LIN {X 0,Y 418.252,Z 144.006,A -85,B 0,C 180,E1 -10131.558,E2 -10131.558} C_VEL
LIN {X 0,Y 418.26,Z 144.01,A -85,B 0,C 180,E1 -10135.159,E2 -10135.159} C_VEL
LIN {X 0,Y 418.268,Z 144.145,A -85,B 0,C 180,E1 -10137.972,E2 -10137.972} C_VEL
LIN {X 0,Y 421.832,Z 158.166,A -85,B 0,C 180,E1 -10140.894,E2 -10140.894} C_VEL
LIN {X 0,Y 424.172,Z 168.884,A -85,B 0,C 180,E1 -10142.964,E2 -10142.964} C_VEL
LIN {X 0,Y 426.899,Z 180.828,A -85,B 0,C 180,E1 -10143.399,E2 -10143.399} C_VEL
LIN {X 0,Y 430.73,Z 200.296,A -85,B 0,C 180,E1 -10144.007,E2 -10144.007} C_VEL
LIN {X 0,Y 428.4,Z 334.091,A -85,B 0,C 180,E1 -10146.301,E2 -10146.301} C_VEL
LIN {X 0,Y 427.722,Z 349.611,A -85,B 0,C 180,E1 -10146.742,E2 -10146.742} C_VEL
LIN {X 0,Y 426.907,Z 363.658,A -85,B 0,C 180,E1 -10147.324,E2 -10147.324} C_VEL
LIN {X 0,Y 425.923,Z 377.546,A -85,B 0,C 180,E1 -10148.079,E2 -10148.079} C_VEL
LIN {X 0,Y 424.665,Z 391.423,A -85,B 0,C 180,E1 -10149.03,E2 -10149.03} C_VEL
LIN {X 0,Y 423.505,Z 404.135,A -85,B 0,C 180,E1 -10150.111,E2 -10150.111} C_VEL
LIN {X 0,Y 422.222,Z 416.989,A -85,B 0,C 180,E1 -10151.437,E2 -10151.437} C_VEL
LIN {X 0,Y 421.112,Z 427.749,A -85,B 0,C 180,E1 -10152.768,E2 -10152.768} C_VEL
LIN {X 0,Y 420.039,Z 437.702,A -85,B 0,C 180,E1 -10154.223,E2 -10154.223} C_VEL
LIN {X 0,Y 419.06,Z 447.438,A -85,B 0,C 180,E1 -10155.926,E2 -10155.926} C_VEL
LIN {X 0,Y 418.334,Z 455.561,A -85,B 0,C 180,E1 -10157.631,E2 -10157.631} C_VEL
LIN {X 0,Y 417.774,Z 462.273,A -85,B 0,C 180,E1 -10159.336,E2 -10159.336} C_VEL
LIN {X 0,Y 417.406,Z 468.473,A -85,B 0,C 180,E1 -10161.284,E2 -10161.284} C_VEL
LIN {X 0,Y 417.166,Z 473.266,A -85,B 0,C 180,E1 -10163.227,E2 -10163.227} C_VEL
LIN {X 0,Y 417.051,Z 476.778,A -85,B 0,C 180,E1 -10165.167,E2 -10165.167} C_VEL
LIN {X 0,Y 416.969,Z 479.087,A -85,B 0,C 180,E1 -10167.102,E2 -10167.102} C_VEL
LIN {X 0,Y 416.989,Z 480.248,A -85,B 0,C 180,E1 -10169.034,E2 -10169.034} C_VEL
LIN {X 0,Y 416.989,Z 480.247,A -85,B 0,C 180,E1 -10170.966,E2 -10170.966} C_VEL
LIN {X 0,Y 416.969,Z 479.078,A -85,B 0,C 180,E1 -10172.898,E2 -10172.898} C_VEL
LIN {X 0,Y 417.055,Z 476.766,A -85,B 0,C 180,E1 -10174.833,E2 -10174.833} C_VEL
LIN {X 0,Y 417.224,Z 473.257,A -85,B 0,C 180,E1 -10176.772,E2 -10176.772} C_VEL
LIN {X 0,Y 417.406,Z 468.462,A -85,B 0,C 180,E1 -10178.716,E2 -10178.716} C_VEL
LIN {X 0,Y 417.774,Z 462.25,A -85,B 0,C 180,E1 -10180.664,E2 -10180.664} C_VEL
LIN {X 0,Y 418.325,Z 455.532,A -85,B 0,C 180,E1 -10182.369,E2 -10182.369} C_VEL
LIN {X 0,Y 419.17,Z 446.15,A -85,B 0,C 180,E1 -10184.318,E2 -10184.318} C_VEL
LIN {X 0,Y 420.2,Z 436.15,A -85,B 0,C 180,E1 -10186.02,E2 -10186.02} C_VEL
LIN {X 0,Y 421.313,Z 425.92,A -85,B 0,C 180,E1 -10187.473,E2 -10187.473} C_VEL
LIN {X 0,Y 422.432,Z 414.801,A -85,B 0,C 180,E1 -10188.805,E2 -10188.805} C_VEL
LIN {X 0,Y 423.625,Z 402.782,A -85,B 0,C 180,E1 -10190.009,E2 -10190.009} C_VEL
LIN {X 0,Y 424.808,Z 389.749,A -85,B 0,C 180,E1 -10191.09,E2 -10191.09} C_VEL
LIN {X 0,Y 426.096,Z 375.444,A -85,B 0,C 180,E1 -10192.039,E2 -10192.039} C_VEL
LIN {X 0,Y 427.014,Z 361.163,A -85,B 0,C 180,E1 -10192.786,E2 -10192.786} C_VEL
LIN {X 0,Y 427.86,Z 345.756,A -85,B 0,C 180,E1 -10193.378,E2 -10193.378} C_VEL
LIN {X 0,Y 428.437,Z 330.738,A -85,B 0,C 180,E1 -10193.761,E2 -10193.761} C_VEL
LIN {X 0,Y 430.681,Z 199.743,A -85,B 0,C 180,E1 -10195.998,E2 -10195.998} C_VEL
LIN {X 0,Y 424.482,Z 170.317,A -85,B 0,C 180,E1 -10196.951,E2 -10196.951} C_VEL
LIN {X 0,Y 424.129,Z 168.838,A -85,B 0,C 180,E1 -10197.034,E2 -10197.034} C_VEL
LIN {X 0,Y 421.815,Z 158.115,A -85,B 0,C 180,E1 -10199.108,E2 -10199.108} C_VEL
LIN {X 0,Y 418.268,Z 144.112,A -85,B 0,C 180,E1 -10202.028,E2 -10202.028} C_VEL
LIN {X 0,Y 418.259,Z 144.01,A -85,B 0,C 180,E1 -10204.841,E2 -10204.841} C_VEL
LIN {X 0,Y 418.251,Z 144.005,A -85,B 0,C 180,E1 -10208.442,E2 -10208.442} C_VEL
LIN {X 0,Y 418.24,Z 144.008,A -85,B 0,C 180,E1 -10212.233,E2 -10212.233} C_VEL
LIN {X 0,Y 418.236,Z 144.004,A -85,B 0,C 180,E1 -10215.109,E2 -10215.109} C_VEL
LIN {X 0,Y 418.24,Z 144.004,A -85,B 0,C 180,E1 -10217.767,E2 -10217.767} C_VEL
LIN {X 0,Y 418.253,Z 143.996,A -85,B 0,C 180,E1 -10220.62,E2 -10220.62} C_VEL
LIN {X 0,Y 418.243,Z 144.006,A -85,B 0,C 180,E1 -10223.976,E2 -10223.976} C_VEL
LIN {X 0,Y 418.243,Z 143.976,A -85,B 0,C 180,E1 -10227.472,E2 -10227.472} C_VEL
LIN {X 0,Y 418.269,Z 144.006,A -85,B 0,C 180,E1 -10230.896,E2 -10230.896} C_VEL
LIN {X 0,Y 418.27,Z 143.998,A -85,B 0,C 180,E1 -10234.096,E2 -10234.096} C_VEL
LIN {X 0,Y 418.239,Z 144.01,A -85,B 0,C 180,E1 -10237.264,E2 -10237.264} C_VEL
LIN {X 0,Y 418.284,Z 144,A -85,B 0,C 180,E1 -10240.364,E2 -10240.364} C_VEL
LIN {X 0,Y 418.317,Z 143.993,A -85,B 0,C 180,E1 -10243.405,E2 -10243.405} C_VEL
LIN {X 0,Y 418.348,Z 144.002,A -85,B 0,C 180,E1 -10246.999,E2 -10246.999} C_VEL
LIN {X 0,Y 418.34,Z 143.986,A -85,B 0,C 180,E1 -10250.329,E2 -10250.329} C_VEL
LIN {X 0,Y 418.462,Z 143.982,A -85,B 0,C 180,E1 -10253.249,E2 -10253.249} C_VEL
LIN {X 0,Y 418.334,Z 143.989,A -85,B 0,C 180,E1 -10255.182,E2 -10255.182} C_VEL
LIN {X 0,Y 418.543,Z 143.966,A -85,B 0,C 180,E1 -10258.076,E2 -10258.076} C_VEL
LIN {X 0,Y 418.668,Z 143.956,A -85,B 0,C 180,E1 -10260,E2 -10260} C_VEL
LIN {X 0,Y 418.488,Z 143.969,A -85,B 0,C 180,E1 -10262.888,E2 -10262.888} C_VEL
LIN {X 0,Y 418.459,Z 143.979,A -85,B 0,C 180,E1 -10266.516,E2 -10266.516} C_VEL
LIN {X 0,Y 418.34,Z 143.99,A -85,B 0,C 180,E1 -10269.672,E2 -10269.672} C_VEL
LIN {X 0,Y 418.348,Z 143.992,A -85,B 0,C 180,E1 -10273.001,E2 -10273.001} C_VEL
LIN {X 0,Y 418.306,Z 144.002,A -85,B 0,C 180,E1 -10276.732,E2 -10276.732} C_VEL
LIN {X 0,Y 418.272,Z 143.998,A -85,B 0,C 180,E1 -10279.79,E2 -10279.79} C_VEL
LIN {X 0,Y 418.229,Z 144.011,A -85,B 0,C 180,E1 -10282.737,E2 -10282.737} C_VEL
LIN {X 0,Y 418.226,Z 144.007,A -85,B 0,C 180,E1 -10285.907,E2 -10285.907} C_VEL
LIN {X 0,Y 418.26,Z 144.007,A -85,B 0,C 180,E1 -10289.162,E2 -10289.162} C_VEL
LIN {X 0,Y 418.251,Z 143.974,A -85,B 0,C 180,E1 -10292.842,E2 -10292.842} C_VEL
LIN {X 0,Y 418.244,Z 144.011,A -85,B 0,C 180,E1 -10296.238,E2 -10296.238} C_VEL
LIN {X 0,Y 418.2,Z 143.987,A -85,B 0,C 180,E1 -10299.688,E2 -10299.688} C_VEL
LIN {X 0,Y 418.208,Z 144.011,A -85,B 0,C 180,E1 -10302.318,E2 -10302.318} C_VEL
LIN {X 0,Y 418.236,Z 144.002,A -85,B 0,C 180,E1 -10305.109,E2 -10305.109} C_VEL
LIN {X 0,Y 418.219,Z 144.015,A -85,B 0,C 180,E1 -10307.764,E2 -10307.764} C_VEL
LIN {X 0,Y 418.238,Z 144.013,A -85,B 0,C 180,E1 -10311.557,E2 -10311.557} C_VEL
LIN {X 0,Y 418.251,Z 144.014,A -85,B 0,C 180,E1 -10315.158,E2 -10315.158} C_VEL
LIN {X 0,Y 418.24,Z 144.014,A -85,B 0,C 180,E1 -10317.471,E2 -10317.471} C_VEL
LIN {X 0,Y 418.236,Z 144.048,A -85,B 0,C 180,E1 -10319.072,E2 -10319.072} C_VEL
LIN {X 0,Y 418.652,Z 145.744,A -85,B 0,C 180,E1 -10319.519,E2 -10319.519} C_VEL
LIN {X 0,Y 421.734,Z 158.326,A -85,B 0,C 180,E1 -10322.186,E2 -10322.186} C_VEL
LIN {X 0,Y 422.604,Z 162.134,A -85,B 0,C 180,E1 -10322.921,E2 -10322.921} C_VEL
LIN {X 0,Y 426.969,Z 173.061,A -85,B 0,C 180,E1 -10323.446,E2 -10323.446} C_VEL
LIN {X 0,Y 430.77,Z 191.061,A -85,B 0,C 180,E1 -10324.027,E2 -10324.027} C_VEL
LIN {X 0,Y 428.844,Z 307.257,A -85,B 0,C 180,E1 -10326.006,E2 -10326.006} C_VEL
LIN {X 0,Y 428.375,Z 329.622,A -85,B 0,C 180,E1 -10326.428,E2 -10326.428} C_VEL
LIN {X 0,Y 427.679,Z 344.966,A -85,B 0,C 180,E1 -10326.901,E2 -10326.901} C_VEL
LIN {X 0,Y 426.893,Z 359.501,A -85,B 0,C 180,E1 -10327.544,E2 -10327.544} C_VEL
LIN {X 0,Y 425.872,Z 373.217,A -85,B 0,C 180,E1 -10328.331,E2 -10328.331} C_VEL
LIN {X 0,Y 424.685,Z 386.502,A -85,B 0,C 180,E1 -10329.284,E2 -10329.284} C_VEL
LIN {X 0,Y 423.406,Z 400.005,A -85,B 0,C 180,E1 -10330.485,E2 -10330.485} C_VEL
LIN {X 0,Y 422.251,Z 411.523,A -85,B 0,C 180,E1 -10331.727,E2 -10331.727} C_VEL
LIN {X 0,Y 421.139,Z 421.713,A -85,B 0,C 180,E1 -10333.03,E2 -10333.03} C_VEL
LIN {X 0,Y 420.108,Z 425.828,A -85,B 0,C 180,E1 -10333.591,E2 -10333.591} C_VEL
LIN {X 0,Y 416.611,Z 432.311,A -85,B 0,C 180,E1 -10334.503,E2 -10334.503} C_VEL
LIN {X 0,Y 413.133,Z 438.422,A -85,B 0,C 180,E1 -10335.477,E2 -10335.477} C_VEL
LIN {X 0,Y 412.145,Z 441.818,A -85,B 0,C 180,E1 -10336.129,E2 -10336.129} C_VEL
LIN {X 0,Y 411.461,Z 449.785,A -85,B 0,C 180,E1 -10337.922,E2 -10337.922} C_VEL
LIN {X 0,Y 410.786,Z 456.159,A -85,B 0,C 180,E1 -10339.651,E2 -10339.651} C_VEL
LIN {X 0,Y 410.382,Z 462.015,A -85,B 0,C 180,E1 -10341.63,E2 -10341.63} C_VEL
LIN {X 0,Y 410.106,Z 466.665,A -85,B 0,C 180,E1 -10343.694,E2 -10343.694} C_VEL
LIN {X 0,Y 410.013,Z 468.998,A -85,B 0,C 180,E1 -10345.083,E2 -10345.083} C_VEL
LIN {X 0,Y 409.92,Z 471.324,A -85,B 0,C 180,E1 -10347.052,E2 -10347.052} C_VEL
LIN {X 0,Y 409.917,Z 472.513,A -85,B 0,C 180,E1 -10349.018,E2 -10349.018} C_VEL
LIN {X 0,Y 409.917,Z 472.529,A -85,B 0,C 180,E1 -10350.982,E2 -10350.982} C_VEL
LIN {X 0,Y 409.92,Z 471.405,A -85,B 0,C 180,E1 -10352.948,E2 -10352.948} C_VEL
LIN {X 0,Y 410.004,Z 469.143,A -85,B 0,C 180,E1 -10354.917,E2 -10354.917} C_VEL
LIN {X 0,Y 410.113,Z 465.687,A -85,B 0,C 180,E1 -10356.89,E2 -10356.89} C_VEL
LIN {X 0,Y 410.441,Z 460.957,A -85,B 0,C 180,E1 -10358.865,E2 -10358.865} C_VEL
LIN {X 0,Y 410.894,Z 454.829,A -85,B 0,C 180,E1 -10360.845,E2 -10360.845} C_VEL
LIN {X 0,Y 411.543,Z 448.17,A -85,B 0,C 180,E1 -10362.576,E2 -10362.576} C_VEL
LIN {X 0,Y 412.45,Z 438.891,A -85,B 0,C 180,E1 -10364.557,E2 -10364.557} C_VEL
LIN {X 0,Y 413.564,Z 428.987,A -85,B 0,C 180,E1 -10366.284,E2 -10366.284} C_VEL
LIN {X 0,Y 414.74,Z 418.833,A -85,B 0,C 180,E1 -10367.759,E2 -10367.759} C_VEL
LIN {X 0,Y 416.013,Z 406.748,A -85,B 0,C 180,E1 -10369.234,E2 -10369.234} C_VEL
LIN {X 0,Y 417.297,Z 394.633,A -85,B 0,C 180,E1 -10370.455,E2 -10370.455} C_VEL
LIN {X 0,Y 418.547,Z 381.471,A -85,B 0,C 180,E1 -10371.55,E2 -10371.55} C_VEL
LIN {X 0,Y 419.642,Z 368.934,A -85,B 0,C 180,E1 -10372.396,E2 -10372.396} C_VEL
LIN {X 0,Y 420.635,Z 354.753,A -85,B 0,C 180,E1 -10373.16,E2 -10373.16} C_VEL
LIN {X 0,Y 421.407,Z 340.861,A -85,B 0,C 180,E1 -10373.725,E2 -10373.725} C_VEL
LIN {X 0,Y 422.025,Z 325.906,A -85,B 0,C 180,E1 -10374.145,E2 -10374.145} C_VEL
LIN {X 0,Y 424.493,Z 192.916,A -85,B 0,C 180,E1 -10376.453,E2 -10376.453} C_VEL
LIN {X 0,Y 420.689,Z 174.699,A -85,B 0,C 180,E1 -10377.053,E2 -10377.053} C_VEL
LIN {X 0,Y 415.364,Z 162.13,A -85,B 0,C 180,E1 -10377.699,E2 -10377.699} C_VEL
LIN {X 0,Y 412.224,Z 148.968,A -85,B 0,C 180,E1 -10380.479,E2 -10380.479} C_VEL
LIN {X 0,Y 411.237,Z 145.352,A -85,B 0,C 180,E1 -10381.296,E2 -10381.296} C_VEL
LIN {X 0,Y 411.152,Z 144.881,A -85,B 0,C 180,E1 -10381.594,E2 -10381.594} C_VEL
LIN {X 0,Y 411.202,Z 144.891,A -85,B 0,C 180,E1 -10384.876,E2 -10384.876} C_VEL
LIN {X 0,Y 411.191,Z 144.891,A -85,B 0,C 180,E1 -10388.166,E2 -10388.166} C_VEL
LIN {X 0,Y 411.161,Z 144.894,A -85,B 0,C 180,E1 -10391.808,E2 -10391.808} C_VEL
LIN {X 0,Y 411.174,Z 144.89,A -85,B 0,C 180,E1 -10395.509,E2 -10395.509} C_VEL
LIN {X 0,Y 411.148,Z 144.874,A -85,B 0,C 180,E1 -10398.775,E2 -10398.775} C_VEL
LIN {X 0,Y 411.186,Z 144.88,A -85,B 0,C 180,E1 -10402.025,E2 -10402.025} C_VEL
LIN {X 0,Y 411.204,Z 144.881,A -85,B 0,C 180,E1 -10405.123,E2 -10405.123} C_VEL
LIN {X 0,Y 411.164,Z 144.853,A -85,B 0,C 180,E1 -10408.002,E2 -10408.002} C_VEL
LIN {X 0,Y 411.177,Z 144.888,A -85,B 0,C 180,E1 -10411.407,E2 -10411.407} C_VEL
LIN {X 0,Y 411.19,Z 144.879,A -85,B 0,C 180,E1 -10414.941,E2 -10414.941} C_VEL
LIN {X 0,Y 411.205,Z 144.89,A -85,B 0,C 180,E1 -10417.913,E2 -10417.913} C_VEL
LIN {X 0,Y 411.217,Z 144.879,A -85,B 0,C 180,E1 -10421.051,E2 -10421.051} C_VEL
LIN {X 0,Y 411.212,Z 144.882,A -85,B 0,C 180,E1 -10424.13,E2 -10424.13} C_VEL
LIN {X 0,Y 411.305,Z 144.869,A -85,B 0,C 180,E1 -10427.166,E2 -10427.166} C_VEL
LIN {X 0,Y 411.292,Z 144.869,A -85,B 0,C 180,E1 -10430.161,E2 -10430.161} C_VEL
LIN {X 0,Y 411.426,Z 144.854,A -85,B 0,C 180,E1 -10433.132,E2 -10433.132} C_VEL
LIN {X 0,Y 411.3,Z 144.875,A -85,B 0,C 180,E1 -10435.099,E2 -10435.099} C_VEL
LIN {X 0,Y 411.507,Z 144.838,A -85,B 0,C 180,E1 -10438.042,E2 -10438.042} C_VEL
LIN {X 0,Y 411.636,Z 144.833,A -85,B 0,C 180,E1 -10440,E2 -10440} C_VEL
LIN {X 0,Y 411.451,Z 144.847,A -85,B 0,C 180,E1 -10442.937,E2 -10442.937} C_VEL
LIN {X 0,Y 411.426,Z 144.859,A -85,B 0,C 180,E1 -10446.867,E2 -10446.867} C_VEL
LIN {X 0,Y 411.293,Z 144.864,A -85,B 0,C 180,E1 -10449.839,E2 -10449.839} C_VEL
LIN {X 0,Y 411.308,Z 144.878,A -85,B 0,C 180,E1 -10453.104,E2 -10453.104} C_VEL
LIN {X 0,Y 411.259,Z 144.875,A -85,B 0,C 180,E1 -10456.889,E2 -10456.889} C_VEL
LIN {X 0,Y 411.232,Z 144.878,A -85,B 0,C 180,E1 -10459.987,E2 -10459.987} C_VEL
LIN {X 0,Y 411.197,Z 144.891,A -85,B 0,C 180,E1 -10463.148,E2 -10463.148} C_VEL
LIN {X 0,Y 411.235,Z 144.874,A -85,B 0,C 180,E1 -10466.381,E2 -10466.381} C_VEL
LIN {X 0,Y 411.202,Z 144.884,A -85,B 0,C 180,E1 -10469.712,E2 -10469.712} C_VEL
LIN {X 0,Y 411.205,Z 144.85,A -85,B 0,C 180,E1 -10473.156,E2 -10473.156} C_VEL
LIN {X 0,Y 411.193,Z 144.891,A -85,B 0,C 180,E1 -10476.552,E2 -10476.552} C_VEL
LIN {X 0,Y 411.213,Z 144.866,A -85,B 0,C 180,E1 -10479.728,E2 -10479.728} C_VEL
LIN {X 0,Y 411.174,Z 144.892,A -85,B 0,C 180,E1 -10483.133,E2 -10483.133} C_VEL
LIN {X 0,Y 411.168,Z 144.876,A -85,B 0,C 180,E1 -10485.881,E2 -10485.881} C_VEL
LIN {X 0,Y 411.164,Z 144.892,A -85,B 0,C 180,E1 -10488.771,E2 -10488.771} C_VEL
LIN {X 0,Y 411.196,Z 144.89,A -85,B 0,C 180,E1 -10492.026,E2 -10492.026} C_VEL
LIN {X 0,Y 411.207,Z 144.89,A -85,B 0,C 180,E1 -10495.666,E2 -10495.666} C_VEL
LIN {X 0,Y 411.224,Z 145.01,A -85,B 0,C 180,E1 -10497.537,E2 -10497.537} C_VEL
LIN {X 0,Y 414.354,Z 157.383,A -85,B 0,C 180,E1 -10500.184,E2 -10500.184} C_VEL
LIN {X 0,Y 417.031,Z 168.833,A -85,B 0,C 180,E1 -10502.464,E2 -10502.464} C_VEL
LIN {X 0,Y 418.721,Z 173.884,A -85,B 0,C 180,E1 -10502.707,E2 -10502.707} C_VEL
LIN {X 0,Y 424.313,Z 200.872,A -85,B 0,C 180,E1 -10503.596,E2 -10503.596} C_VEL
LIN {X 0,Y 421.943,Z 332.536,A -85,B 0,C 180,E1 -10505.883,E2 -10505.883} C_VEL
LIN {X 0,Y 421.314,Z 347.724,A -85,B 0,C 180,E1 -10506.302,E2 -10506.302} C_VEL
LIN {X 0,Y 420.419,Z 362.017,A -85,B 0,C 180,E1 -10506.875,E2 -10506.875} C_VEL
LIN {X 0,Y 419.503,Z 375.496,A -85,B 0,C 180,E1 -10507.596,E2 -10507.596} C_VEL
LIN {X 0,Y 418.209,Z 389.779,A -85,B 0,C 180,E1 -10508.561,E2 -10508.561} C_VEL
LIN {X 0,Y 416.935,Z 402.78,A -85,B 0,C 180,E1 -10509.656,E2 -10509.656} C_VEL
LIN {X 0,Y 415.649,Z 414.783,A -85,B 0,C 180,E1 -10510.877,E2 -10510.877} C_VEL
LIN {X 0,Y 414.492,Z 425.899,A -85,B 0,C 180,E1 -10512.23,E2 -10512.23} C_VEL
LIN {X 0,Y 413.326,Z 436.124,A -85,B 0,C 180,E1 -10513.706,E2 -10513.706} C_VEL
LIN {X 0,Y 412.275,Z 446.117,A -85,B 0,C 180,E1 -10515.437,E2 -10515.437} C_VEL
LIN {X 0,Y 411.337,Z 455.495,A -85,B 0,C 180,E1 -10517.418,E2 -10517.418} C_VEL
LIN {X 0,Y 410.763,Z 462.208,A -85,B 0,C 180,E1 -10519.152,E2 -10519.152} C_VEL
LIN {X 0,Y 410.331,Z 468.407,A -85,B 0,C 180,E1 -10521.133,E2 -10521.133} C_VEL
LIN {X 0,Y 410.082,Z 473.2,A -85,B 0,C 180,E1 -10523.11,E2 -10523.11} C_VEL
LIN {X 0,Y 409.963,Z 476.712,A -85,B 0,C 180,E1 -10525.083,E2 -10525.083} C_VEL
LIN {X 0,Y 409.867,Z 479.02,A -85,B 0,C 180,E1 -10527.051,E2 -10527.051} C_VEL
LIN {X 0,Y 409.915,Z 480.182,A -85,B 0,C 180,E1 -10529.018,E2 -10529.018} C_VEL
LIN {X 0,Y 409.915,Z 480.181,A -85,B 0,C 180,E1 -10530.982,E2 -10530.982} C_VEL
LIN {X 0,Y 409.867,Z 479.012,A -85,B 0,C 180,E1 -10532.949,E2 -10532.949} C_VEL
LIN {X 0,Y 409.968,Z 476.699,A -85,B 0,C 180,E1 -10534.917,E2 -10534.917} C_VEL
LIN {X 0,Y 410.155,Z 473.19,A -85,B 0,C 180,E1 -10536.889,E2 -10536.889} C_VEL
LIN {X 0,Y 410.331,Z 468.394,A -85,B 0,C 180,E1 -10538.867,E2 -10538.867} C_VEL
LIN {X 0,Y 410.763,Z 462.183,A -85,B 0,C 180,E1 -10540.848,E2 -10540.848} C_VEL
LIN {X 0,Y 411.33,Z 455.464,A -85,B 0,C 180,E1 -10542.583,E2 -10542.583} C_VEL
LIN {X 0,Y 412.263,Z 446.081,A -85,B 0,C 180,E1 -10544.563,E2 -10544.563} C_VEL
LIN {X 0,Y 413.301,Z 436.081,A -85,B 0,C 180,E1 -10546.295,E2 -10546.295} C_VEL
LIN {X 0,Y 414.588,Z 424.669,A -85,B 0,C 180,E1 -10547.926,E2 -10547.926} C_VEL
LIN {X 0,Y 415.901,Z 412.51,A -85,B 0,C 180,E1 -10549.368,E2 -10549.368} C_VEL
LIN {X 0,Y 417.212,Z 400.083,A -85,B 0,C 180,E1 -10550.588,E2 -10550.588} C_VEL
LIN {X 0,Y 418.48,Z 386.466,A -85,B 0,C 180,E1 -10551.683,E2 -10551.683} C_VEL
LIN {X 0,Y 419.708,Z 372.359,A -85,B 0,C 180,E1 -10552.587,E2 -10552.587} C_VEL
LIN {X 0,Y 420.673,Z 358.594,A -85,B 0,C 180,E1 -10553.274,E2 -10553.274} C_VEL
LIN {X 0,Y 421.505,Z 342.93,A -85,B 0,C 180,E1 -10553.849,E2 -10553.849} C_VEL
LIN {X 0,Y 422.007,Z 327.643,A -85,B 0,C 180,E1 -10554.211,E2 -10554.211} C_VEL
LIN {X 0,Y 424.332,Z 201.581,A -85,B 0,C 180,E1 -10556.381,E2 -10556.381} C_VEL
LIN {X 0,Y 419.585,Z 177.878,A -85,B 0,C 180,E1 -10557.147,E2 -10557.147} C_VEL
LIN {X 0,Y 417.817,Z 171.092,A -85,B 0,C 180,E1 -10557.4,E2 -10557.4} C_VEL
LIN {X 0,Y 416.985,Z 168.667,A -85,B 0,C 180,E1 -10557.548,E2 -10557.548} C_VEL
LIN {X 0,Y 414.1,Z 156.176,A -85,B 0,C 180,E1 -10560.054,E2 -10560.054} C_VEL
LIN {X 0,Y 411.224,Z 144.948,A -85,B 0,C 180,E1 -10562.481,E2 -10562.481} C_VEL
LIN {X 0,Y 411.198,Z 144.881,A -85,B 0,C 180,E1 -10565.529,E2 -10565.529} C_VEL
LIN {X 0,Y 411.212,Z 144.874,A -85,B 0,C 180,E1 -10569.225,E2 -10569.225} C_VEL
LIN {X 0,Y 411.182,Z 144.885,A -85,B 0,C 180,E1 -10572.696,E2 -10572.696} C_VEL
LIN {X 0,Y 411.168,Z 144.893,A -85,B 0,C 180,E1 -10575.881,E2 -10575.881} C_VEL
LIN {X 0,Y 411.163,Z 144.873,A -85,B 0,C 180,E1 -10578.772,E2 -10578.772} C_VEL
LIN {X 0,Y 411.205,Z 144.885,A -85,B 0,C 180,E1 -10581.832,E2 -10581.832} C_VEL
LIN {X 0,Y 411.203,Z 144.87,A -85,B 0,C 180,E1 -10585.123,E2 -10585.123} C_VEL
LIN {X 0,Y 411.164,Z 144.862,A -85,B 0,C 180,E1 -10588.003,E2 -10588.003} C_VEL
LIN {X 0,Y 411.219,Z 144.889,A -85,B 0,C 180,E1 -10591.41,E2 -10591.41} C_VEL
LIN {X 0,Y 411.238,Z 144.874,A -85,B 0,C 180,E1 -10593.619,E2 -10593.619} C_VEL
LIN {X 0,Y 411.204,Z 144.89,A -85,B 0,C 180,E1 -10596.853,E2 -10596.853} C_VEL
LIN {X 0,Y 411.216,Z 144.88,A -85,B 0,C 180,E1 -10600.051,E2 -10600.051} C_VEL
LIN {X 0,Y 411.264,Z 144.874,A -85,B 0,C 180,E1 -10603.131,E2 -10603.131} C_VEL
LIN {X 0,Y 411.307,Z 144.878,A -85,B 0,C 180,E1 -10606.896,E2 -10606.896} C_VEL
LIN {X 0,Y 411.292,Z 144.864,A -85,B 0,C 180,E1 -10610.161,E2 -10610.161} C_VEL
LIN {X 0,Y 411.426,Z 144.859,A -85,B 0,C 180,E1 -10613.133,E2 -10613.133} C_VEL
LIN {X 0,Y 411.305,Z 144.865,A -85,B 0,C 180,E1 -10615.099,E2 -10615.099} C_VEL
LIN {X 0,Y 411.511,Z 144.842,A -85,B 0,C 180,E1 -10618.043,E2 -10618.043} C_VEL
LIN {X 0,Y 411.637,Z 144.832,A -85,B 0,C 180,E1 -10620,E2 -10620} C_VEL
LIN {X 0,Y 411.445,Z 144.846,A -85,B 0,C 180,E1 -10622.937,E2 -10622.937} C_VEL
LIN {X 0,Y 411.424,Z 144.855,A -85,B 0,C 180,E1 -10626.514,E2 -10626.514} C_VEL
LIN {X 0,Y 411.292,Z 144.869,A -85,B 0,C 180,E1 -10629.839,E2 -10629.839} C_VEL
LIN {X 0,Y 411.307,Z 144.869,A -85,B 0,C 180,E1 -10633.104,E2 -10633.104} C_VEL
LIN {X 0,Y 411.258,Z 144.879,A -85,B 0,C 180,E1 -10636.889,E2 -10636.889} C_VEL
LIN {X 0,Y 411.232,Z 144.874,A -85,B 0,C 180,E1 -10639.987,E2 -10639.987} C_VEL
LIN {X 0,Y 411.19,Z 144.888,A -85,B 0,C 180,E1 -10643.148,E2 -10643.148} C_VEL
LIN {X 0,Y 411.176,Z 144.889,A -85,B 0,C 180,E1 -10646.385,E2 -10646.385} C_VEL
LIN {X 0,Y 411.198,Z 144.876,A -85,B 0,C 180,E1 -10649.713,E2 -10649.713} C_VEL
LIN {X 0,Y 411.205,Z 144.854,A -85,B 0,C 180,E1 -10653.156,E2 -10653.156} C_VEL
LIN {X 0,Y 411.192,Z 144.889,A -85,B 0,C 180,E1 -10656.552,E2 -10656.552} C_VEL
LIN {X 0,Y 411.169,Z 144.862,A -85,B 0,C 180,E1 -10659.72,E2 -10659.72} C_VEL
LIN {X 0,Y 411.163,Z 144.894,A -85,B 0,C 180,E1 -10663.135,E2 -10663.135} C_VEL
LIN {X 0,Y 411.164,Z 144.876,A -85,B 0,C 180,E1 -10665.882,E2 -10665.882} C_VEL
LIN {X 0,Y 411.148,Z 144.896,A -85,B 0,C 180,E1 -10668.774,E2 -10668.774} C_VEL
LIN {X 0,Y 411.186,Z 144.891,A -85,B 0,C 180,E1 -10672.025,E2 -10672.025} C_VEL
LIN {X 0,Y 411.203,Z 144.892,A -85,B 0,C 180,E1 -10675.123,E2 -10675.123} C_VEL
LIN {X 0,Y 411.153,Z 144.882,A -85,B 0,C 180,E1 -10678.405,E2 -10678.405} C_VEL
LIN {X 0,Y 411.218,Z 145.209,A -85,B 0,C 180,E1 -10678.763,E2 -10678.763} C_VEL
LIN {X 0,Y 414.2,Z 156.981,A -85,B 0,C 180,E1 -10681.358,E2 -10681.358} C_VEL
LIN {X 0,Y 415.438,Z 162.329,A -85,B 0,C 180,E1 -10682.423,E2 -10682.423} C_VEL
LIN {X 0,Y 420.788,Z 175.035,A -85,B 0,C 180,E1 -10683.06,E2 -10683.06} C_VEL
LIN {X 0,Y 424.408,Z 192.602,A -85,B 0,C 180,E1 -10683.634,E2 -10683.634} C_VEL
LIN {X 0,Y 422.385,Z 307.349,A -85,B 0,C 180,E1 -10685.616,E2 -10685.616} C_VEL
LIN {X 0,Y 421.877,Z 329.705,A -85,B 0,C 180,E1 -10686.042,E2 -10686.042} C_VEL
LIN {X 0,Y 421.187,Z 344.47,A -85,B 0,C 180,E1 -10686.499,E2 -10686.499} C_VEL
LIN {X 0,Y 420.4,Z 358.732,A -85,B 0,C 180,E1 -10687.129,E2 -10687.129} C_VEL
LIN {X 0,Y 419.42,Z 371.398,A -85,B 0,C 180,E1 -10687.851,E2 -10687.851} C_VEL
LIN {X 0,Y 418.161,Z 385.01,A -85,B 0,C 180,E1 -10688.817,E2 -10688.817} C_VEL
LIN {X 0,Y 416.821,Z 398.82,A -85,B 0,C 180,E1 -10690.036,E2 -10690.036} C_VEL
LIN {X 0,Y 415.605,Z 410.212,A -85,B 0,C 180,E1 -10691.259,E2 -10691.259} C_VEL
LIN {X 0,Y 414.324,Z 421.713,A -85,B 0,C 180,E1 -10692.732,E2 -10692.732} C_VEL
LIN {X 0,Y 413.292,Z 431.392,A -85,B 0,C 180,E1 -10694.212,E2 -10694.212} C_VEL
LIN {X 0,Y 412.229,Z 440.881,A -85,B 0,C 180,E1 -10695.94,E2 -10695.94} C_VEL
LIN {X 0,Y 412.145,Z 441.818,A -85,B 0,C 180,E1 -10696.129,E2 -10696.129} C_VEL
LIN {X 0,Y 411.184,Z 445.107,A -85,B 0,C 180,E1 -10696.8,E2 -10696.8} C_VEL
LIN {X 0,Y 407.838,Z 450.165,A -85,B 0,C 180,E1 -10697.9,E2 -10697.9} C_VEL
LIN {X 0,Y 404.548,Z 454.796,A -85,B 0,C 180,E1 -10699.055,E2 -10699.055} C_VEL
LIN {X 0,Y 403.691,Z 457.295,A -85,B 0,C 180,E1 -10699.804,E2 -10699.804} C_VEL
LIN {X 0,Y 403.32,Z 462.082,A -85,B 0,C 180,E1 -10701.482,E2 -10701.482} C_VEL
LIN {X 0,Y 403.076,Z 465.55,A -85,B 0,C 180,E1 -10702.99,E2 -10702.99} C_VEL
LIN {X 0,Y 402.928,Z 469.065,A -85,B 0,C 180,E1 -10704.997,E2 -10704.997} C_VEL
LIN {X 0,Y 402.819,Z 471.391,A -85,B 0,C 180,E1 -10707,E2 -10707} C_VEL
LIN {X 0,Y 402.845,Z 472.579,A -85,B 0,C 180,E1 -10709,E2 -10709} C_VEL
LIN {X 0,Y 402.846,Z 472.595,A -85,B 0,C 180,E1 -10711,E2 -10711} C_VEL
LIN {X 0,Y 402.819,Z 471.472,A -85,B 0,C 180,E1 -10713,E2 -10713} C_VEL
LIN {X 0,Y 402.917,Z 469.209,A -85,B 0,C 180,E1 -10715.003,E2 -10715.003} C_VEL
LIN {X 0,Y 403.048,Z 465.753,A -85,B 0,C 180,E1 -10717.011,E2 -10717.011} C_VEL
LIN {X 0,Y 403.403,Z 461.022,A -85,B 0,C 180,E1 -10719.021,E2 -10719.021} C_VEL
LIN {X 0,Y 403.889,Z 454.894,A -85,B 0,C 180,E1 -10721.035,E2 -10721.035} C_VEL
LIN {X 0,Y 404.538,Z 448.235,A -85,B 0,C 180,E1 -10722.797,E2 -10722.797} C_VEL
LIN {X 0,Y 405.515,Z 438.955,A -85,B 0,C 180,E1 -10724.811,E2 -10724.811} C_VEL
LIN {X 0,Y 406.713,Z 429.051,A -85,B 0,C 180,E1 -10726.566,E2 -10726.566} C_VEL
LIN {X 0,Y 407.946,Z 418.897,A -85,B 0,C 180,E1 -10728.065,E2 -10728.065} C_VEL
LIN {X 0,Y 409.148,Z 407.879,A -85,B 0,C 180,E1 -10729.439,E2 -10729.439} C_VEL
LIN {X 0,Y 410.483,Z 395.984,A -85,B 0,C 180,E1 -10730.679,E2 -10730.679} C_VEL
LIN {X 0,Y 411.774,Z 383.112,A -85,B 0,C 180,E1 -10731.791,E2 -10731.791} C_VEL
LIN {X 0,Y 413.082,Z 368.993,A -85,B 0,C 180,E1 -10732.772,E2 -10732.772} C_VEL
LIN {X 0,Y 414.153,Z 354.057,A -85,B 0,C 180,E1 -10733.582,E2 -10733.582} C_VEL
LIN {X 0,Y 414.966,Z 339.085,A -85,B 0,C 180,E1 -10734.183,E2 -10734.183} C_VEL
LIN {X 0,Y 415.583,Z 324.447,A -85,B 0,C 180,E1 -10734.577,E2 -10734.577} C_VEL
LIN {X 0,Y 418.139,Z 194.125,A -85,B 0,C 180,E1 -10736.865,E2 -10736.865} C_VEL
LIN {X 0,Y 414.702,Z 177.431,A -85,B 0,C 180,E1 -10737.425,E2 -10737.425} C_VEL
LIN {X 0,Y 408.159,Z 162.135,A -85,B 0,C 180,E1 -10738.237,E2 -10738.237} C_VEL
LIN {X 0,Y 404.958,Z 149.039,A -85,B 0,C 180,E1 -10741.085,E2 -10741.085} C_VEL
LIN {X 0,Y 404.148,Z 145.977,A -85,B 0,C 180,E1 -10741.822,E2 -10741.822} C_VEL
LIN {X 0,Y 404.138,Z 145.762,A -85,B 0,C 180,E1 -10743.813,E2 -10743.813} C_VEL
LIN {X 0,Y 404.132,Z 145.761,A -85,B 0,C 180,E1 -10746.874,E2 -10746.874} C_VEL
LIN {X 0,Y 404.118,Z 145.757,A -85,B 0,C 180,E1 -10750.075,E2 -10750.075} C_VEL
LIN {X 0,Y 404.142,Z 145.758,A -85,B 0,C 180,E1 -10753.082,E2 -10753.082} C_VEL
LIN {X 0,Y 404.121,Z 145.768,A -85,B 0,C 180,E1 -10755.922,E2 -10755.922} C_VEL
LIN {X 0,Y 404.102,Z 145.753,A -85,B 0,C 180,E1 -10758.633,E2 -10758.633} C_VEL
LIN {X 0,Y 404.14,Z 145.752,A -85,B 0,C 180,E1 -10761.495,E2 -10761.495} C_VEL
LIN {X 0,Y 404.179,Z 145.757,A -85,B 0,C 180,E1 -10764.983,E2 -10764.983} C_VEL
LIN {X 0,Y 404.138,Z 145.729,A -85,B 0,C 180,E1 -10768.443,E2 -10768.443} C_VEL
LIN {X 0,Y 404.152,Z 145.761,A -85,B 0,C 180,E1 -10770.862,E2 -10770.862} C_VEL
LIN {X 0,Y 404.155,Z 145.755,A -85,B 0,C 180,E1 -10774.722,E2 -10774.722} C_VEL
LIN {X 0,Y 404.168,Z 145.763,A -85,B 0,C 180,E1 -10777.508,E2 -10777.508} C_VEL
LIN {X 0,Y 404.162,Z 145.757,A -85,B 0,C 180,E1 -10780.707,E2 -10780.707} C_VEL
LIN {X 0,Y 404.183,Z 145.761,A -85,B 0,C 180,E1 -10783.846,E2 -10783.846} C_VEL
LIN {X 0,Y 404.285,Z 145.743,A -85,B 0,C 180,E1 -10786.939,E2 -10786.939} C_VEL
LIN {X 0,Y 404.258,Z 145.747,A -85,B 0,C 180,E1 -10789.988,E2 -10789.988} C_VEL
LIN {X 0,Y 404.371,Z 145.732,A -85,B 0,C 180,E1 -10793.012,E2 -10793.012} C_VEL
LIN {X 0,Y 404.273,Z 145.75,A -85,B 0,C 180,E1 -10795.013,E2 -10795.013} C_VEL
LIN {X 0,Y 404.475,Z 145.713,A -85,B 0,C 180,E1 -10798.008,E2 -10798.008} C_VEL
LIN {X 0,Y 404.605,Z 145.709,A -85,B 0,C 180,E1 -10800,E2 -10800} C_VEL
LIN {X 0,Y 404.409,Z 145.723,A -85,B 0,C 180,E1 -10802.988,E2 -10802.988} C_VEL
LIN {X 0,Y 404.372,Z 145.739,A -85,B 0,C 180,E1 -10806.988,E2 -10806.988} C_VEL
LIN {X 0,Y 404.258,Z 145.741,A -85,B 0,C 180,E1 -10810.012,E2 -10810.012} C_VEL
LIN {X 0,Y 404.268,Z 145.753,A -85,B 0,C 180,E1 -10813.211,E2 -10813.211} C_VEL
LIN {X 0,Y 404.218,Z 145.754,A -85,B 0,C 180,E1 -10817.007,E2 -10817.007} C_VEL
LIN {X 0,Y 404.165,Z 145.758,A -85,B 0,C 180,E1 -10820.351,E2 -10820.351} C_VEL
LIN {X 0,Y 404.161,Z 145.764,A -85,B 0,C 180,E1 -10823.575,E2 -10823.575} C_VEL
LIN {X 0,Y 404.182,Z 145.751,A -85,B 0,C 180,E1 -10825.766,E2 -10825.766} C_VEL
LIN {X 0,Y 404.196,Z 145.759,A -85,B 0,C 180,E1 -10827.999,E2 -10827.999} C_VEL
LIN {X 0,Y 404.139,Z 145.743,A -85,B 0,C 180,E1 -10831.558,E2 -10831.558} C_VEL
LIN {X 0,Y 404.179,Z 145.748,A -85,B 0,C 180,E1 -10835.017,E2 -10835.017} C_VEL
LIN {X 0,Y 404.155,Z 145.754,A -85,B 0,C 180,E1 -10838.757,E2 -10838.757} C_VEL
LIN {X 0,Y 404.123,Z 145.756,A -85,B 0,C 180,E1 -10841.599,E2 -10841.599} C_VEL
LIN {X 0,Y 404.146,Z 145.761,A -85,B 0,C 180,E1 -10844.522,E2 -10844.522} C_VEL
LIN {X 0,Y 404.137,Z 145.762,A -85,B 0,C 180,E1 -10847.295,E2 -10847.295} C_VEL
LIN {X 0,Y 404.169,Z 145.753,A -85,B 0,C 180,E1 -10849.955,E2 -10849.955} C_VEL
LIN {X 0,Y 404.138,Z 145.765,A -85,B 0,C 180,E1 -10853.125,E2 -10853.125} C_VEL
LIN {X 0,Y 404.146,Z 145.755,A -85,B 0,C 180,E1 -10856.188,E2 -10856.188} C_VEL
LIN {X 0,Y 404.224,Z 145.982,A -85,B 0,C 180,E1 -10857.119,E2 -10857.119} C_VEL
LIN {X 0,Y 407.179,Z 157.584,A -85,B 0,C 180,E1 -10859.656,E2 -10859.656} C_VEL
LIN {X 0,Y 409.765,Z 168.645,A -85,B 0,C 180,E1 -10861.922,E2 -10861.922} C_VEL
LIN {X 0,Y 412.564,Z 175.812,A -85,B 0,C 180,E1 -10862.303,E2 -10862.303} C_VEL
LIN {X 0,Y 417.739,Z 200.965,A -85,B 0,C 180,E1 -10863.15,E2 -10863.15} C_VEL
LIN {X 0,Y 417.943,Z 204.055,A -85,B 0,C 180,E1 -10863.222,E2 -10863.222} C_VEL
LIN {X 0,Y 415.445,Z 333.991,A -85,B 0,C 180,E1 -10865.514,E2 -10865.514} C_VEL
LIN {X 0,Y 414.7,Z 349.498,A -85,B 0,C 180,E1 -10865.967,E2 -10865.967} C_VEL
LIN {X 0,Y 413.793,Z 363.539,A -85,B 0,C 180,E1 -10866.563,E2 -10866.563} C_VEL
LIN {X 0,Y 412.754,Z 377.424,A -85,B 0,C 180,E1 -10867.341,E2 -10867.341} C_VEL
LIN {X 0,Y 411.41,Z 391.299,A -85,B 0,C 180,E1 -10868.32,E2 -10868.32} C_VEL
LIN {X 0,Y 410.102,Z 404.009,A -85,B 0,C 180,E1 -10869.432,E2 -10869.432} C_VEL
LIN {X 0,Y 408.686,Z 416.861,A -85,B 0,C 180,E1 -10870.799,E2 -10870.799} C_VEL
LIN {X 0,Y 407.469,Z 427.62,A -85,B 0,C 180,E1 -10872.172,E2 -10872.172} C_VEL
LIN {X 0,Y 406.289,Z 437.572,A -85,B 0,C 180,E1 -10873.674,E2 -10873.674} C_VEL
LIN {X 0,Y 405.175,Z 447.307,A -85,B 0,C 180,E1 -10875.433,E2 -10875.433} C_VEL
LIN {X 0,Y 404.36,Z 455.43,A -85,B 0,C 180,E1 -10877.197,E2 -10877.197} C_VEL
LIN {X 0,Y 403.764,Z 462.143,A -85,B 0,C 180,E1 -10878.961,E2 -10878.961} C_VEL
LIN {X 0,Y 403.277,Z 468.341,A -85,B 0,C 180,E1 -10880.976,E2 -10880.976} C_VEL
LIN {X 0,Y 403.002,Z 473.134,A -85,B 0,C 180,E1 -10882.988,E2 -10882.988} C_VEL
LIN {X 0,Y 402.879,Z 476.646,A -85,B 0,C 180,E1 -10884.996,E2 -10884.996} C_VEL
LIN {X 0,Y 402.769,Z 478.954,A -85,B 0,C 180,E1 -10886.999,E2 -10886.999} C_VEL
LIN {X 0,Y 402.842,Z 480.116,A -85,B 0,C 180,E1 -10889,E2 -10889} C_VEL
LIN {X 0,Y 402.842,Z 480.115,A -85,B 0,C 180,E1 -10891,E2 -10891} C_VEL
LIN {X 0,Y 402.769,Z 478.945,A -85,B 0,C 180,E1 -10893.001,E2 -10893.001} C_VEL
LIN {X 0,Y 402.883,Z 476.632,A -85,B 0,C 180,E1 -10895.004,E2 -10895.004} C_VEL
LIN {X 0,Y 403.065,Z 473.123,A -85,B 0,C 180,E1 -10897.011,E2 -10897.011} C_VEL
LIN {X 0,Y 403.277,Z 468.326,A -85,B 0,C 180,E1 -10899.024,E2 -10899.024} C_VEL
LIN {X 0,Y 403.763,Z 462.115,A -85,B 0,C 180,E1 -10901.038,E2 -10901.038} C_VEL
LIN {X 0,Y 404.354,Z 455.395,A -85,B 0,C 180,E1 -10902.803,E2 -10902.803} C_VEL
LIN {X 0,Y 405.162,Z 447.271,A -85,B 0,C 180,E1 -10904.567,E2 -10904.567} C_VEL
LIN {X 0,Y 406.268,Z 437.529,A -85,B 0,C 180,E1 -10906.326,E2 -10906.326} C_VEL
LIN {X 0,Y 407.474,Z 427.567,A -85,B 0,C 180,E1 -10907.827,E2 -10907.827} C_VEL
LIN {X 0,Y 408.69,Z 416.802,A -85,B 0,C 180,E1 -10909.201,E2 -10909.201} C_VEL
LIN {X 0,Y 410.107,Z 403.935,A -85,B 0,C 180,E1 -10910.567,E2 -10910.567} C_VEL
LIN {X 0,Y 411.382,Z 391.191,A -85,B 0,C 180,E1 -10911.681,E2 -10911.681} C_VEL
LIN {X 0,Y 412.752,Z 377.287,A -85,B 0,C 180,E1 -10912.659,E2 -10912.659} C_VEL
LIN {X 0,Y 413.726,Z 364.28,A -85,B 0,C 180,E1 -10913.395,E2 -10913.395} C_VEL
LIN {X 0,Y 414.728,Z 349.27,A -85,B 0,C 180,E1 -10914.031,E2 -10914.031} C_VEL
LIN {X 0,Y 415.404,Z 333.586,A -85,B 0,C 180,E1 -10914.488,E2 -10914.488} C_VEL
LIN {X 0,Y 417.753,Z 210.809,A -85,B 0,C 180,E1 -10916.654,E2 -10916.654} C_VEL
LIN {X 0,Y 417.863,Z 201.734,A -85,B 0,C 180,E1 -10916.817,E2 -10916.817} C_VEL
LIN {X 0,Y 412.298,Z 174.92,A -85,B 0,C 180,E1 -10917.723,E2 -10917.723} C_VEL
LIN {X 0,Y 409.796,Z 168.717,A -85,B 0,C 180,E1 -10918.058,E2 -10918.058} C_VEL
LIN {X 0,Y 407.182,Z 157.529,A -85,B 0,C 180,E1 -10920.345,E2 -10920.345} C_VEL
LIN {X 0,Y 404.187,Z 145.837,A -85,B 0,C 180,E1 -10922.918,E2 -10922.918} C_VEL
LIN {X 0,Y 404.143,Z 145.759,A -85,B 0,C 180,E1 -10926.246,E2 -10926.246} C_VEL
LIN {X 0,Y 404.152,Z 145.756,A -85,B 0,C 180,E1 -10928.757,E2 -10928.757} C_VEL
LIN {X 0,Y 404.123,Z 145.773,A -85,B 0,C 180,E1 -10931.6,E2 -10931.6} C_VEL
LIN {X 0,Y 404.145,Z 145.753,A -85,B 0,C 180,E1 -10934.522,E2 -10934.522} C_VEL
LIN {X 0,Y 404.136,Z 145.768,A -85,B 0,C 180,E1 -10937.296,E2 -10937.296} C_VEL
LIN {X 0,Y 404.169,Z 145.74,A -85,B 0,C 180,E1 -10939.956,E2 -10939.956} C_VEL
LIN {X 0,Y 404.136,Z 145.77,A -85,B 0,C 180,E1 -10943.125,E2 -10943.125} C_VEL
LIN {X 0,Y 404.138,Z 145.733,A -85,B 0,C 180,E1 -10946.187,E2 -10946.187} C_VEL
LIN {X 0,Y 404.146,Z 145.759,A -85,B 0,C 180,E1 -10949.715,E2 -10949.715} C_VEL
LIN {X 0,Y 404.196,Z 145.754,A -85,B 0,C 180,E1 -10953.123,E2 -10953.123} C_VEL
LIN {X 0,Y 404.179,Z 145.762,A -85,B 0,C 180,E1 -10955.335,E2 -10955.335} C_VEL
LIN {X 0,Y 404.14,Z 145.759,A -85,B 0,C 180,E1 -10958.581,E2 -10958.581} C_VEL
LIN {X 0,Y 404.205,Z 145.758,A -85,B 0,C 180,E1 -10961.762,E2 -10961.762} C_VEL
LIN {X 0,Y 404.207,Z 145.748,A -85,B 0,C 180,E1 -10964.882,E2 -10964.882} C_VEL
LIN {X 0,Y 404.258,Z 145.751,A -85,B 0,C 180,E1 -10967.959,E2 -10967.959} C_VEL
LIN {X 0,Y 404.267,Z 145.741,A -85,B 0,C 180,E1 -10970.999,E2 -10970.999} C_VEL
LIN {X 0,Y 404.395,Z 145.734,A -85,B 0,C 180,E1 -10974.015,E2 -10974.015} C_VEL
LIN {X 0,Y 404.48,Z 145.717,A -85,B 0,C 180,E1 -10978.009,E2 -10978.009} C_VEL
LIN {X 0,Y 404.607,Z 145.708,A -85,B 0,C 180,E1 -10980,E2 -10980} C_VEL
LIN {X 0,Y 404.404,Z 145.723,A -85,B 0,C 180,E1 -10982.989,E2 -10982.989} C_VEL
LIN {X 0,Y 404.373,Z 145.734,A -85,B 0,C 180,E1 -10986.509,E2 -10986.509} C_VEL
LIN {X 0,Y 404.267,Z 145.74,A -85,B 0,C 180,E1 -10989.002,E2 -10989.002} C_VEL
LIN {X 0,Y 404.257,Z 145.756,A -85,B 0,C 180,E1 -10992.042,E2 -10992.042} C_VEL
LIN {X 0,Y 404.198,Z 145.749,A -85,B 0,C 180,E1 -10995.118,E2 -10995.118} C_VEL
LIN {X 0,Y 404.202,Z 145.757,A -85,B 0,C 180,E1 -10998.239,E2 -10998.239} C_VEL
LIN {X 0,Y 404.139,Z 145.762,A -85,B 0,C 180,E1 -11001.419,E2 -11001.419} C_VEL
LIN {X 0,Y 404.149,Z 145.756,A -85,B 0,C 180,E1 -11004.668,E2 -11004.668} C_VEL
LIN {X 0,Y 404.117,Z 145.771,A -85,B 0,C 180,E1 -11008.006,E2 -11008.006} C_VEL
LIN {X 0,Y 404.144,Z 145.749,A -85,B 0,C 180,E1 -11010.285,E2 -11010.285} C_VEL
LIN {X 0,Y 404.139,Z 145.742,A -85,B 0,C 180,E1 -11013.813,E2 -11013.813} C_VEL
LIN {X 0,Y 404.135,Z 145.77,A -85,B 0,C 180,E1 -11016.875,E2 -11016.875} C_VEL
LIN {X 0,Y 404.117,Z 145.738,A -85,B 0,C 180,E1 -11020.075,E2 -11020.075} C_VEL
LIN {X 0,Y 404.143,Z 145.767,A -85,B 0,C 180,E1 -11023.082,E2 -11023.082} C_VEL
LIN {X 0,Y 404.121,Z 145.753,A -85,B 0,C 180,E1 -11025.922,E2 -11025.922} C_VEL
LIN {X 0,Y 404.103,Z 145.775,A -85,B 0,C 180,E1 -11028.633,E2 -11028.633} C_VEL
LIN {X 0,Y 404.141,Z 145.767,A -85,B 0,C 180,E1 -11031.495,E2 -11031.495} C_VEL
LIN {X 0,Y 404.174,Z 145.766,A -85,B 0,C 180,E1 -11034.983,E2 -11034.983} C_VEL
LIN {X 0,Y 404.141,Z 145.907,A -85,B 0,C 180,E1 -11038.25,E2 -11038.25} C_VEL
LIN {X 0,Y 406.612,Z 155.688,A -85,B 0,C 180,E1 -11040.498,E2 -11040.498} C_VEL
LIN {X 0,Y 408.209,Z 162.188,A -85,B 0,C 180,E1 -11041.874,E2 -11041.874} C_VEL
LIN {X 0,Y 414.812,Z 177.978,A -85,B 0,C 180,E1 -11042.694,E2 -11042.694} C_VEL
LIN {X 0,Y 418.039,Z 193.082,A -85,B 0,C 180,E1 -11043.208,E2 -11043.208} C_VEL
LIN {X 0,Y 415.95,Z 307.441,A -85,B 0,C 180,E1 -11045.213,E2 -11045.213} C_VEL
LIN {X 0,Y 415.405,Z 329.787,A -85,B 0,C 180,E1 -11045.645,E2 -11045.645} C_VEL
LIN {X 0,Y 414.67,Z 344.721,A -85,B 0,C 180,E1 -11046.115,E2 -11046.115} C_VEL
LIN {X 0,Y 413.844,Z 359.189,A -85,B 0,C 180,E1 -11046.768,E2 -11046.768} C_VEL
LIN {X 0,Y 412.85,Z 371.472,A -85,B 0,C 180,E1 -11047.479,E2 -11047.479} C_VEL
LIN {X 0,Y 411.55,Z 385.083,A -85,B 0,C 180,E1 -11048.46,E2 -11048.46} C_VEL
LIN {X 0,Y 410.245,Z 397.602,A -85,B 0,C 180,E1 -11049.571,E2 -11049.571} C_VEL
LIN {X 0,Y 408.961,Z 409.216,A -85,B 0,C 180,E1 -11050.812,E2 -11050.812} C_VEL
LIN {X 0,Y 407.755,Z 420.004,A -85,B 0,C 180,E1 -11052.186,E2 -11052.186} C_VEL
LIN {X 0,Y 406.572,Z 429.98,A -85,B 0,C 180,E1 -11053.686,E2 -11053.686} C_VEL
LIN {X 0,Y 405.422,Z 439.723,A -85,B 0,C 180,E1 -11055.442,E2 -11055.442} C_VEL
LIN {X 0,Y 404.629,Z 447.844,A -85,B 0,C 180,E1 -11057.206,E2 -11057.206} C_VEL
LIN {X 0,Y 403.913,Z 454.546,A -85,B 0,C 180,E1 -11058.966,E2 -11058.966} C_VEL
LIN {X 0,Y 403.691,Z 457.295,A -85,B 0,C 180,E1 -11059.804,E2 -11059.804} C_VEL
LIN {X 0,Y 402.872,Z 459.669,A -85,B 0,C 180,E1 -11060.564,E2 -11060.564} C_VEL
LIN {X 0,Y 399.767,Z 463.197,A -85,B 0,C 180,E1 -11061.811,E2 -11061.811} C_VEL
LIN {X 0,Y 397.172,Z 465.6,A -85,B 0,C 180,E1 -11062.839,E2 -11062.839} C_VEL
LIN {X 0,Y 396.02,Z 467.14,A -85,B 0,C 180,E1 -11063.651,E2 -11063.651} C_VEL
LIN {X 0,Y 395.904,Z 467.596,A -85,B 0,C 180,E1 -11063.929,E2 -11063.929} C_VEL
LIN {X 0,Y 395.765,Z 470.439,A -85,B 0,C 180,E1 -11065.927,E2 -11065.927} C_VEL
LIN {X 0,Y 395.759,Z 472.191,A -85,B 0,C 180,E1 -11067.965,E2 -11067.965} C_VEL
LIN {X 0,Y 395.758,Z 472.804,A -85,B 0,C 180,E1 -11070,E2 -11070} C_VEL
LIN {X 0,Y 395.759,Z 472.239,A -85,B 0,C 180,E1 -11072.035,E2 -11072.035} C_VEL
LIN {X 0,Y 395.762,Z 470.551,A -85,B 0,C 180,E1 -11074.073,E2 -11074.073} C_VEL
LIN {X 0,Y 395.859,Z 467.61,A -85,B 0,C 180,E1 -11076.167,E2 -11076.167} C_VEL
LIN {X 0,Y 396.157,Z 463.619,A -85,B 0,C 180,E1 -11078.159,E2 -11078.159} C_VEL
LIN {X 0,Y 396.587,Z 458.208,A -85,B 0,C 180,E1 -11080.207,E2 -11080.207} C_VEL
LIN {X 0,Y 397.342,Z 451.314,A -85,B 0,C 180,E1 -11082.254,E2 -11082.254} C_VEL
LIN {X 0,Y 398.167,Z 442.713,A -85,B 0,C 180,E1 -11084.307,E2 -11084.307} C_VEL
LIN {X 0,Y 399.282,Z 433.569,A -85,B 0,C 180,E1 -11086.095,E2 -11086.095} C_VEL
LIN {X 0,Y 400.427,Z 424.252,A -85,B 0,C 180,E1 -11087.623,E2 -11087.623} C_VEL
LIN {X 0,Y 401.627,Z 414.737,A -85,B 0,C 180,E1 -11088.944,E2 -11088.944} C_VEL
LIN {X 0,Y 403.081,Z 402.253,A -85,B 0,C 180,E1 -11090.409,E2 -11090.409} C_VEL
LIN {X 0,Y 404.539,Z 389.209,A -85,B 0,C 180,E1 -11091.665,E2 -11091.665} C_VEL
LIN {X 0,Y 405.831,Z 376.516,A -85,B 0,C 180,E1 -11092.663,E2 -11092.663} C_VEL
LIN {X 0,Y 407.173,Z 361.888,A -85,B 0,C 180,E1 -11093.578,E2 -11093.578} C_VEL
LIN {X 0,Y 408.09,Z 346.999,A -85,B 0,C 180,E1 -11094.296,E2 -11094.296} C_VEL
LIN {X 0,Y 408.884,Z 332.087,A -85,B 0,C 180,E1 -11094.803,E2 -11094.803} C_VEL
LIN {X 0,Y 409.409,Z 312.806,A -85,B 0,C 180,E1 -11095.21,E2 -11095.21} C_VEL
LIN {X 0,Y 411.784,Z 194.551,A -85,B 0,C 180,E1 -11097.307,E2 -11097.307} C_VEL
LIN {X 0,Y 408.541,Z 179.759,A -85,B 0,C 180,E1 -11097.83,E2 -11097.83} C_VEL
LIN {X 0,Y 401.065,Z 162.507,A -85,B 0,C 180,E1 -11098.76,E2 -11098.76} C_VEL
LIN {X 0,Y 400.195,Z 159.061,A -85,B 0,C 180,E1 -11099.454,E2 -11099.454} C_VEL
LIN {X 0,Y 397.142,Z 147.052,A -85,B 0,C 180,E1 -11102.216,E2 -11102.216} C_VEL
LIN {X 0,Y 397.107,Z 146.648,A -85,B 0,C 180,E1 -11102.519,E2 -11102.519} C_VEL
LIN {X 0,Y 397.093,Z 146.64,A -85,B 0,C 180,E1 -11105.736,E2 -11105.736} C_VEL
LIN {X 0,Y 397.092,Z 146.641,A -85,B 0,C 180,E1 -11108.854,E2 -11108.854} C_VEL
LIN {X 0,Y 397.055,Z 146.652,A -85,B 0,C 180,E1 -11112.269,E2 -11112.269} C_VEL
LIN {X 0,Y 397.085,Z 146.635,A -85,B 0,C 180,E1 -11115.069,E2 -11115.069} C_VEL
LIN {X 0,Y 397.052,Z 146.643,A -85,B 0,C 180,E1 -11118.024,E2 -11118.024} C_VEL
LIN {X 0,Y 397.092,Z 146.634,A -85,B 0,C 180,E1 -11121.724,E2 -11121.724} C_VEL
LIN {X 0,Y 397.121,Z 146.634,A -85,B 0,C 180,E1 -11125.506,E2 -11125.506} C_VEL
LIN {X 0,Y 397.077,Z 146.616,A -85,B 0,C 180,E1 -11129.117,E2 -11129.117} C_VEL
LIN {X 0,Y 397.08,Z 146.649,A -85,B 0,C 180,E1 -11132.247,E2 -11132.247} C_VEL
LIN {X 0,Y 397.105,Z 146.632,A -85,B 0,C 180,E1 -11134.865,E2 -11134.865} C_VEL
LIN {X 0,Y 397.097,Z 146.644,A -85,B 0,C 180,E1 -11138.181,E2 -11138.181} C_VEL
LIN {X 0,Y 397.153,Z 146.631,A -85,B 0,C 180,E1 -11141.426,E2 -11141.426} C_VEL
LIN {X 0,Y 397.127,Z 146.631,A -85,B 0,C 180,E1 -11144.606,E2 -11144.606} C_VEL
LIN {X 0,Y 397.221,Z 146.628,A -85,B 0,C 180,E1 -11147.742,E2 -11147.742} C_VEL
LIN {X 0,Y 397.237,Z 146.616,A -85,B 0,C 180,E1 -11150.838,E2 -11150.838} C_VEL
LIN {X 0,Y 397.358,Z 146.615,A -85,B 0,C 180,E1 -11153.908,E2 -11153.908} C_VEL
LIN {X 0,Y 397.444,Z 146.588,A -85,B 0,C 180,E1 -11157.973,E2 -11157.973} C_VEL
LIN {X 0,Y 397.575,Z 146.584,A -85,B 0,C 180,E1 -11160,E2 -11160} C_VEL
LIN {X 0,Y 397.343,Z 146.602,A -85,B 0,C 180,E1 -11163.042,E2 -11163.042} C_VEL
LIN {X 0,Y 397.347,Z 146.612,A -85,B 0,C 180,E1 -11166.092,E2 -11166.092} C_VEL
LIN {X 0,Y 397.237,Z 146.615,A -85,B 0,C 180,E1 -11169.162,E2 -11169.162} C_VEL
LIN {X 0,Y 397.221,Z 146.628,A -85,B 0,C 180,E1 -11172.258,E2 -11172.258} C_VEL
LIN {X 0,Y 397.18,Z 146.622,A -85,B 0,C 180,E1 -11175.392,E2 -11175.392} C_VEL
LIN {X 0,Y 397.159,Z 146.638,A -85,B 0,C 180,E1 -11178.573,E2 -11178.573} C_VEL
LIN {X 0,Y 397.097,Z 146.638,A -85,B 0,C 180,E1 -11181.818,E2 -11181.818} C_VEL
LIN {X 0,Y 397.152,Z 146.627,A -85,B 0,C 180,E1 -11185.512,E2 -11185.512} C_VEL
LIN {X 0,Y 397.124,Z 146.644,A -85,B 0,C 180,E1 -11188.543,E2 -11188.543} C_VEL
LIN {X 0,Y 397.077,Z 146.612,A -85,B 0,C 180,E1 -11192.072,E2 -11192.072} C_VEL
LIN {X 0,Y 397.117,Z 146.636,A -85,B 0,C 180,E1 -11195.502,E2 -11195.502} C_VEL
LIN {X 0,Y 397.13,Z 146.627,A -85,B 0,C 180,E1 -11198.861,E2 -11198.861} C_VEL
LIN {X 0,Y 397.069,Z 146.641,A -85,B 0,C 180,E1 -11202.267,E2 -11202.267} C_VEL
LIN {X 0,Y 397.087,Z 146.635,A -85,B 0,C 180,E1 -11205.069,E2 -11205.069} C_VEL
LIN {X 0,Y 397.067,Z 146.649,A -85,B 0,C 180,E1 -11208.021,E2 -11208.021} C_VEL
LIN {X 0,Y 397.128,Z 146.631,A -85,B 0,C 180,E1 -11211.139,E2 -11211.139} C_VEL
LIN {X 0,Y 397.12,Z 146.634,A -85,B 0,C 180,E1 -11214.496,E2 -11214.496} C_VEL
LIN {X 0,Y 397.158,Z 146.848,A -85,B 0,C 180,E1 -11216.648,E2 -11216.648} C_VEL
LIN {X 0,Y 400.541,Z 160.075,A -85,B 0,C 180,E1 -11219.6,E2 -11219.6} C_VEL
LIN {X 0,Y 402.612,Z 168.691,A -85,B 0,C 180,E1 -11221.388,E2 -11221.388} C_VEL
LIN {X 0,Y 406.545,Z 178.331,A -85,B 0,C 180,E1 -11221.907,E2 -11221.907} C_VEL
LIN {X 0,Y 411.56,Z 202.985,A -85,B 0,C 180,E1 -11222.753,E2 -11222.753} C_VEL
LIN {X 0,Y 409.49,Z 310.202,A -85,B 0,C 180,E1 -11224.659,E2 -11224.659} C_VEL
LIN {X 0,Y 408.891,Z 336.371,A -85,B 0,C 180,E1 -11225.163,E2 -11225.163} C_VEL
LIN {X 0,Y 408.083,Z 351.63,A -85,B 0,C 180,E1 -11225.645,E2 -11225.645} C_VEL
LIN {X 0,Y 407.22,Z 364.683,A -85,B 0,C 180,E1 -11226.224,E2 -11226.224} C_VEL
LIN {X 0,Y 406.026,Z 379.35,A -85,B 0,C 180,E1 -11227.079,E2 -11227.079} C_VEL
LIN {X 0,Y 404.64,Z 392.819,A -85,B 0,C 180,E1 -11228.073,E2 -11228.073} C_VEL
LIN {X 0,Y 403.136,Z 406.53,A -85,B 0,C 180,E1 -11229.327,E2 -11229.327} C_VEL
LIN {X 0,Y 401.648,Z 419.219,A -85,B 0,C 180,E1 -11230.75,E2 -11230.75} C_VEL
LIN {X 0,Y 400.214,Z 431.104,A -85,B 0,C 180,E1 -11232.367,E2 -11232.367} C_VEL
LIN {X 0,Y 398.87,Z 441.919,A -85,B 0,C 180,E1 -11234.151,E2 -11234.151} C_VEL
LIN {X 0,Y 397.822,Z 451.021,A -85,B 0,C 180,E1 -11235.963,E2 -11235.963} C_VEL
LIN {X 0,Y 397.173,Z 458.395,A -85,B 0,C 180,E1 -11237.74,E2 -11237.74} C_VEL
LIN {X 0,Y 396.401,Z 465.361,A -85,B 0,C 180,E1 -11239.788,E2 -11239.788} C_VEL
LIN {X 0,Y 396.06,Z 470.839,A -85,B 0,C 180,E1 -11241.839,E2 -11241.839} C_VEL
LIN {X 0,Y 395.859,Z 474.979,A -85,B 0,C 180,E1 -11243.885,E2 -11243.885} C_VEL
LIN {X 0,Y 395.732,Z 477.88,A -85,B 0,C 180,E1 -11245.926,E2 -11245.926} C_VEL
LIN {X 0,Y 395.714,Z 479.61,A -85,B 0,C 180,E1 -11247.964,E2 -11247.964} C_VEL
LIN {X 0,Y 395.757,Z 480.203,A -85,B 0,C 180,E1 -11250,E2 -11250} C_VEL
LIN {X 0,Y 395.714,Z 479.605,A -85,B 0,C 180,E1 -11252.036,E2 -11252.036} C_VEL
LIN {X 0,Y 395.733,Z 477.867,A -85,B 0,C 180,E1 -11254.074,E2 -11254.074} C_VEL
LIN {X 0,Y 395.896,Z 474.783,A -85,B 0,C 180,E1 -11256.218,E2 -11256.218} C_VEL
LIN {X 0,Y 396.054,Z 470.825,A -85,B 0,C 180,E1 -11258.161,E2 -11258.161} C_VEL
LIN {X 0,Y 396.392,Z 465.338,A -85,B 0,C 180,E1 -11260.212,E2 -11260.212} C_VEL
LIN {X 0,Y 397.146,Z 458.358,A -85,B 0,C 180,E1 -11262.26,E2 -11262.26} C_VEL
LIN {X 0,Y 397.812,Z 451,A -85,B 0,C 180,E1 -11264.033,E2 -11264.033} C_VEL
LIN {X 0,Y 398.872,Z 441.877,A -85,B 0,C 180,E1 -11265.849,E2 -11265.849} C_VEL
LIN {X 0,Y 400.222,Z 431.049,A -85,B 0,C 180,E1 -11267.633,E2 -11267.633} C_VEL
LIN {X 0,Y 401.641,Z 419.192,A -85,B 0,C 180,E1 -11269.246,E2 -11269.246} C_VEL
LIN {X 0,Y 403.137,Z 406.451,A -85,B 0,C 180,E1 -11270.672,E2 -11270.672} C_VEL
LIN {X 0,Y 404.61,Z 392.705,A -85,B 0,C 180,E1 -11271.929,E2 -11271.929} C_VEL
LIN {X 0,Y 406.034,Z 379.202,A -85,B 0,C 180,E1 -11272.92,E2 -11272.92} C_VEL
LIN {X 0,Y 407.141,Z 365.203,A -85,B 0,C 180,E1 -11273.743,E2 -11273.743} C_VEL
LIN {X 0,Y 408.186,Z 350.074,A -85,B 0,C 180,E1 -11274.408,E2 -11274.408} C_VEL
LIN {X 0,Y 408.917,Z 334.894,A -85,B 0,C 180,E1 -11274.869,E2 -11274.869} C_VEL
LIN {X 0,Y 411.321,Z 215.439,A -85,B 0,C 180,E1 -11277.014,E2 -11277.014} C_VEL
LIN {X 0,Y 411.531,Z 202.925,A -85,B 0,C 180,E1 -11277.239,E2 -11277.239} C_VEL
LIN {X 0,Y 406.351,Z 177.724,A -85,B 0,C 180,E1 -11278.108,E2 -11278.108} C_VEL
LIN {X 0,Y 402.605,Z 168.599,A -85,B 0,C 180,E1 -11278.61,E2 -11278.61} C_VEL
LIN {X 0,Y 399.189,Z 154.586,A -85,B 0,C 180,E1 -11281.585,E2 -11281.585} C_VEL
LIN {X 0,Y 397.135,Z 146.687,A -85,B 0,C 180,E1 -11283.41,E2 -11283.41} C_VEL
LIN {X 0,Y 397.1,Z 146.643,A -85,B 0,C 180,E1 -11286.995,E2 -11286.995} C_VEL
LIN {X 0,Y 397.113,Z 146.629,A -85,B 0,C 180,E1 -11289.577,E2 -11289.577} C_VEL
LIN {X 0,Y 397.102,Z 146.627,A -85,B 0,C 180,E1 -11293.479,E2 -11293.479} C_VEL
LIN {X 0,Y 397.102,Z 146.645,A -85,B 0,C 180,E1 -11296.521,E2 -11296.521} C_VEL
LIN {X 0,Y 397.114,Z 146.623,A -85,B 0,C 180,E1 -11300.423,E2 -11300.423} C_VEL
LIN {X 0,Y 397.106,Z 146.637,A -85,B 0,C 180,E1 -11304.265,E2 -11304.265} C_VEL
LIN {X 0,Y 397.112,Z 146.602,A -85,B 0,C 180,E1 -11306.727,E2 -11306.727} C_VEL
LIN {X 0,Y 397.125,Z 146.638,A -85,B 0,C 180,E1 -11310.296,E2 -11310.296} C_VEL
LIN {X 0,Y 397.195,Z 146.631,A -85,B 0,C 180,E1 -11312.61,E2 -11312.61} C_VEL
LIN {X 0,Y 397.134,Z 146.639,A -85,B 0,C 180,E1 -11315.982,E2 -11315.982} C_VEL
LIN {X 0,Y 397.14,Z 146.633,A -85,B 0,C 180,E1 -11319.705,E2 -11319.705} C_VEL
LIN {X 0,Y 397.183,Z 146.632,A -85,B 0,C 180,E1 -11322.845,E2 -11322.845} C_VEL
LIN {X 0,Y 397.23,Z 146.628,A -85,B 0,C 180,E1 -11326.703,E2 -11326.703} C_VEL
LIN {X 0,Y 397.218,Z 146.617,A -85,B 0,C 180,E1 -11329.809,E2 -11329.809} C_VEL
LIN {X 0,Y 397.32,Z 146.619,A -85,B 0,C 180,E1 -11332.888,E2 -11332.888} C_VEL
LIN {X 0,Y 397.247,Z 146.617,A -85,B 0,C 180,E1 -11334.925,E2 -11334.925} C_VEL
LIN {X 0,Y 397.449,Z 146.593,A -85,B 0,C 180,E1 -11337.973,E2 -11337.973} C_VEL
LIN {X 0,Y 397.576,Z 146.584,A -85,B 0,C 180,E1 -11340,E2 -11340} C_VEL
LIN {X 0,Y 397.337,Z 146.603,A -85,B 0,C 180,E1 -11343.042,E2 -11343.042} C_VEL
LIN {X 0,Y 397.327,Z 146.613,A -85,B 0,C 180,E1 -11346.502,E2 -11346.502} C_VEL
LIN {X 0,Y 397.237,Z 146.616,A -85,B 0,C 180,E1 -11349.162,E2 -11349.162} C_VEL
LIN {X 0,Y 397.22,Z 146.629,A -85,B 0,C 180,E1 -11352.258,E2 -11352.258} C_VEL
LIN {X 0,Y 397.173,Z 146.625,A -85,B 0,C 180,E1 -11355.392,E2 -11355.392} C_VEL
LIN {X 0,Y 397.156,Z 146.631,A -85,B 0,C 180,E1 -11358.574,E2 -11358.574} C_VEL
LIN {X 0,Y 397.096,Z 146.643,A -85,B 0,C 180,E1 -11361.819,E2 -11361.819} C_VEL
LIN {X 0,Y 397.097,Z 146.634,A -85,B 0,C 180,E1 -11365.136,E2 -11365.136} C_VEL
LIN {X 0,Y 397.07,Z 146.645,A -85,B 0,C 180,E1 -11368.548,E2 -11368.548} C_VEL
LIN {X 0,Y 397.08,Z 146.605,A -85,B 0,C 180,E1 -11371.836,E2 -11371.836} C_VEL
LIN {X 0,Y 397.12,Z 146.631,A -85,B 0,C 180,E1 -11374.494,E2 -11374.494} C_VEL
LIN {X 0,Y 397.093,Z 146.636,A -85,B 0,C 180,E1 -11378.276,E2 -11378.276} C_VEL
LIN {X 0,Y 397.052,Z 146.639,A -85,B 0,C 180,E1 -11381.976,E2 -11381.976} C_VEL
LIN {X 0,Y 397.085,Z 146.635,A -85,B 0,C 180,E1 -11385.069,E2 -11385.069} C_VEL
LIN {X 0,Y 397.052,Z 146.651,A -85,B 0,C 180,E1 -11388.024,E2 -11388.024} C_VEL
LIN {X 0,Y 397.093,Z 146.648,A -85,B 0,C 180,E1 -11391.724,E2 -11391.724} C_VEL
LIN {X 0,Y 397.118,Z 146.643,A -85,B 0,C 180,E1 -11395.506,E2 -11395.506} C_VEL
LIN {X 0,Y 397.113,Z 146.774,A -85,B 0,C 180,E1 -11397.782,E2 -11397.782} C_VEL
LIN {X 0,Y 399.583,Z 156.421,A -85,B 0,C 180,E1 -11400.062,E2 -11400.062} C_VEL
LIN {X 0,Y 401.07,Z 162.393,A -85,B 0,C 180,E1 -11401.338,E2 -11401.338} C_VEL
LIN {X 0,Y 408.788,Z 180.394,A -85,B 0,C 180,E1 -11402.302,E2 -11402.302} C_VEL
LIN {X 0,Y 411.68,Z 194.188,A -85,B 0,C 180,E1 -11402.78,E2 -11402.78} C_VEL
LIN {X 0,Y 409.715,Z 296.806,A -85,B 0,C 180,E1 -11404.606,E2 -11404.606} C_VEL
LIN {X 0,Y 408.999,Z 328.729,A -85,B 0,C 180,E1 -11405.204,E2 -11405.204} C_VEL
LIN {X 0,Y 408.263,Z 344.031,A -85,B 0,C 180,E1 -11405.682,E2 -11405.682} C_VEL
LIN {X 0,Y 407.385,Z 358.072,A -85,B 0,C 180,E1 -11406.308,E2 -11406.308} C_VEL
LIN {X 0,Y 406.287,Z 371.546,A -85,B 0,C 180,E1 -11407.095,E2 -11407.095} C_VEL
LIN {X 0,Y 404.924,Z 385.155,A -85,B 0,C 180,E1 -11408.089,E2 -11408.089} C_VEL
LIN {X 0,Y 403.571,Z 397.673,A -85,B 0,C 180,E1 -11409.218,E2 -11409.218} C_VEL
LIN {X 0,Y 402.231,Z 409.287,A -85,B 0,C 180,E1 -11410.478,E2 -11410.478} C_VEL
LIN {X 0,Y 400.979,Z 420.074,A -85,B 0,C 180,E1 -11411.874,E2 -11411.874} C_VEL
LIN {X 0,Y 399.702,Z 430.049,A -85,B 0,C 180,E1 -11413.398,E2 -11413.398} C_VEL
LIN {X 0,Y 398.507,Z 439.792,A -85,B 0,C 180,E1 -11415.184,E2 -11415.184} C_VEL
LIN {X 0,Y 397.637,Z 447.913,A -85,B 0,C 180,E1 -11416.977,E2 -11416.977} C_VEL
LIN {X 0,Y 396.914,Z 454.614,A -85,B 0,C 180,E1 -11418.769,E2 -11418.769} C_VEL
LIN {X 0,Y 396.366,Z 460.822,A -85,B 0,C 180,E1 -11420.818,E2 -11420.818} C_VEL
LIN {X 0,Y 396.003,Z 465.618,A -85,B 0,C 180,E1 -11422.864,E2 -11422.864} C_VEL
LIN {X 0,Y 395.904,Z 467.596,A -85,B 0,C 180,E1 -11423.929,E2 -11423.929} C_VEL
LIN {X 0,Y 395.16,Z 468.951,A -85,B 0,C 180,E1 -11424.758,E2 -11424.758} C_VEL
LIN {X 0,Y 392.22,Z 470.713,A -85,B 0,C 180,E1 -11426.111,E2 -11426.111} C_VEL
LIN {X 0,Y 389.772,Z 471.761,A -85,B 0,C 180,E1 -11427.212,E2 -11427.212} C_VEL
LIN {X 0,Y 388.725,Z 472.327,A -85,B 0,C 180,E1 -11428.069,E2 -11428.069} C_VEL
LIN {X 0,Y 388.641,Z 472.447,A -85,B 0,C 180,E1 -11428.36,E2 -11428.36} C_VEL
LIN {X 0,Y 388.671,Z 472.87,A -85,B 0,C 180,E1 -11430,E2 -11430} C_VEL
LIN {X 0,Y 388.656,Z 472.305,A -85,B 0,C 180,E1 -11432.073,E2 -11432.073} C_VEL
LIN {X 0,Y 388.688,Z 470.617,A -85,B 0,C 180,E1 -11434.148,E2 -11434.148} C_VEL
LIN {X 0,Y 388.794,Z 467.766,A -85,B 0,C 180,E1 -11436.227,E2 -11436.227} C_VEL
LIN {X 0,Y 389.099,Z 463.684,A -85,B 0,C 180,E1 -11438.308,E2 -11438.308} C_VEL
LIN {X 0,Y 389.543,Z 458.273,A -85,B 0,C 180,E1 -11440.394,E2 -11440.394} C_VEL
LIN {X 0,Y 390.362,Z 451.379,A -85,B 0,C 180,E1 -11442.477,E2 -11442.477} C_VEL
LIN {X 0,Y 391.092,Z 443.991,A -85,B 0,C 180,E1 -11444.3,E2 -11444.3} C_VEL
LIN {X 0,Y 392.252,Z 435.041,A -85,B 0,C 180,E1 -11446.124,E2 -11446.124} C_VEL
LIN {X 0,Y 393.374,Z 425.94,A -85,B 0,C 180,E1 -11447.681,E2 -11447.681} C_VEL
LIN {X 0,Y 394.798,Z 415.434,A -85,B 0,C 180,E1 -11449.196,E2 -11449.196} C_VEL
LIN {X 0,Y 396.27,Z 403.487,A -85,B 0,C 180,E1 -11450.64,E2 -11450.64} C_VEL
LIN {X 0,Y 397.762,Z 390.694,A -85,B 0,C 180,E1 -11451.917,E2 -11451.917} C_VEL
LIN {X 0,Y 399.271,Z 376.576,A -85,B 0,C 180,E1 -11453.057,E2 -11453.057} C_VEL
LIN {X 0,Y 400.619,Z 362.71,A -85,B 0,C 180,E1 -11453.941,E2 -11453.941} C_VEL
LIN {X 0,Y 401.573,Z 348.121,A -85,B 0,C 180,E1 -11454.669,E2 -11454.669} C_VEL
LIN {X 0,Y 402.406,Z 333.276,A -85,B 0,C 180,E1 -11455.196,E2 -11455.196} C_VEL
LIN {X 0,Y 402.942,Z 316.424,A -85,B 0,C 180,E1 -11455.575,E2 -11455.575} C_VEL
LIN {X 0,Y 405.482,Z 196,A -85,B 0,C 180,E1 -11457.74,E2 -11457.74} C_VEL
LIN {X 0,Y 402.546,Z 182.402,A -85,B 0,C 180,E1 -11458.229,E2 -11458.229} C_VEL
LIN {X 0,Y 394.335,Z 163.786,A -85,B 0,C 180,E1 -11459.254,E2 -11459.254} C_VEL
LIN {X 0,Y 393.666,Z 161.976,A -85,B 0,C 180,E1 -11459.42,E2 -11459.42} C_VEL
LIN {X 0,Y 390.567,Z 149.729,A -85,B 0,C 180,E1 -11462.249,E2 -11462.249} C_VEL
LIN {X 0,Y 390.084,Z 147.597,A -85,B 0,C 180,E1 -11462.833,E2 -11462.833} C_VEL
LIN {X 0,Y 390.05,Z 147.514,A -85,B 0,C 180,E1 -11466.484,E2 -11466.484} C_VEL
LIN {X 0,Y 390.036,Z 147.514,A -85,B 0,C 180,E1 -11469.212,E2 -11469.212} C_VEL
LIN {X 0,Y 390.031,Z 147.527,A -85,B 0,C 180,E1 -11472.372,E2 -11472.372} C_VEL
LIN {X 0,Y 390.041,Z 147.517,A -85,B 0,C 180,E1 -11475.354,E2 -11475.354} C_VEL
LIN {X 0,Y 390.015,Z 147.514,A -85,B 0,C 180,E1 -11478.184,E2 -11478.184} C_VEL
LIN {X 0,Y 390.058,Z 147.493,A -85,B 0,C 180,E1 -11480.904,E2 -11480.904} C_VEL
LIN {X 0,Y 390.082,Z 147.514,A -85,B 0,C 180,E1 -11484.793,E2 -11484.793} C_VEL
LIN {X 0,Y 390.022,Z 147.485,A -85,B 0,C 180,E1 -11488.495,E2 -11488.495} C_VEL
LIN {X 0,Y 390.026,Z 147.526,A -85,B 0,C 180,E1 -11492.063,E2 -11492.063} C_VEL
LIN {X 0,Y 390.044,Z 147.513,A -85,B 0,C 180,E1 -11495.517,E2 -11495.517} C_VEL
LIN {X 0,Y 390.057,Z 147.515,A -85,B 0,C 180,E1 -11498.878,E2 -11498.878} C_VEL
LIN {X 0,Y 390.104,Z 147.517,A -85,B 0,C 180,E1 -11502.165,E2 -11502.165} C_VEL
LIN {X 0,Y 390.124,Z 147.5,A -85,B 0,C 180,E1 -11505.392,E2 -11505.392} C_VEL
LIN {X 0,Y 390.173,Z 147.504,A -85,B 0,C 180,E1 -11507.517,E2 -11507.517} C_VEL
LIN {X 0,Y 390.195,Z 147.494,A -85,B 0,C 180,E1 -11510.671,E2 -11510.671} C_VEL
LIN {X 0,Y 390.31,Z 147.491,A -85,B 0,C 180,E1 -11513.798,E2 -11513.798} C_VEL
LIN {X 0,Y 390.412,Z 147.463,A -85,B 0,C 180,E1 -11517.937,E2 -11517.937} C_VEL
LIN {X 0,Y 390.544,Z 147.46,A -85,B 0,C 180,E1 -11520,E2 -11520} C_VEL
LIN {X 0,Y 390.279,Z 147.481,A -85,B 0,C 180,E1 -11523.097,E2 -11523.097} C_VEL
LIN {X 0,Y 390.301,Z 147.489,A -85,B 0,C 180,E1 -11526.202,E2 -11526.202} C_VEL
LIN {X 0,Y 390.195,Z 147.491,A -85,B 0,C 180,E1 -11529.329,E2 -11529.329} C_VEL
LIN {X 0,Y 390.173,Z 147.507,A -85,B 0,C 180,E1 -11532.483,E2 -11532.483} C_VEL
LIN {X 0,Y 390.14,Z 147.499,A -85,B 0,C 180,E1 -11535.677,E2 -11535.677} C_VEL
LIN {X 0,Y 390.104,Z 147.517,A -85,B 0,C 180,E1 -11538.922,E2 -11538.922} C_VEL
LIN {X 0,Y 390.038,Z 147.518,A -85,B 0,C 180,E1 -11542.234,E2 -11542.234} C_VEL
LIN {X 0,Y 390.119,Z 147.503,A -85,B 0,C 180,E1 -11545.743,E2 -11545.743} C_VEL
LIN {X 0,Y 390.06,Z 147.52,A -85,B 0,C 180,E1 -11549.109,E2 -11549.109} C_VEL
LIN {X 0,Y 390.041,Z 147.482,A -85,B 0,C 180,E1 -11552.721,E2 -11552.721} C_VEL
LIN {X 0,Y 390.055,Z 147.517,A -85,B 0,C 180,E1 -11555.825,E2 -11555.825} C_VEL
LIN {X 0,Y 390.07,Z 147.503,A -85,B 0,C 180,E1 -11559.218,E2 -11559.218} C_VEL
LIN {X 0,Y 390.043,Z 147.517,A -85,B 0,C 180,E1 -11562.374,E2 -11562.374} C_VEL
LIN {X 0,Y 390.045,Z 147.508,A -85,B 0,C 180,E1 -11565.354,E2 -11565.354} C_VEL
LIN {X 0,Y 390.032,Z 147.527,A -85,B 0,C 180,E1 -11568.187,E2 -11568.187} C_VEL
LIN {X 0,Y 390.089,Z 147.505,A -85,B 0,C 180,E1 -11570.907,E2 -11570.907} C_VEL
LIN {X 0,Y 390.086,Z 147.512,A -85,B 0,C 180,E1 -11574.793,E2 -11574.793} C_VEL
LIN {X 0,Y 390.106,Z 147.746,A -85,B 0,C 180,E1 -11576.165,E2 -11576.165} C_VEL
LIN {X 0,Y 393.372,Z 160.307,A -85,B 0,C 180,E1 -11579.045,E2 -11579.045} C_VEL
LIN {X 0,Y 395.445,Z 168.737,A -85,B 0,C 180,E1 -11580.829,E2 -11580.829} C_VEL
LIN {X 0,Y 400.556,Z 180.836,A -85,B 0,C 180,E1 -11581.5,E2 -11581.5} C_VEL
LIN {X 0,Y 405.243,Z 204.028,A -85,B 0,C 180,E1 -11582.314,E2 -11582.314} C_VEL
LIN {X 0,Y 403.017,Z 313.734,A -85,B 0,C 180,E1 -11584.292,E2 -11584.292} C_VEL
LIN {X 0,Y 402.458,Z 336.318,A -85,B 0,C 180,E1 -11584.739,E2 -11584.739} C_VEL
LIN {X 0,Y 401.614,Z 351.647,A -85,B 0,C 180,E1 -11585.23,E2 -11585.23} C_VEL
LIN {X 0,Y 400.642,Z 365.657,A -85,B 0,C 180,E1 -11585.869,E2 -11585.869} C_VEL
LIN {X 0,Y 399.488,Z 379.289,A -85,B 0,C 180,E1 -11586.682,E2 -11586.682} C_VEL
LIN {X 0,Y 398.028,Z 392.756,A -85,B 0,C 180,E1 -11587.689,E2 -11587.689} C_VEL
LIN {X 0,Y 396.462,Z 406.466,A -85,B 0,C 180,E1 -11588.963,E2 -11588.963} C_VEL
LIN {X 0,Y 394.88,Z 419.351,A -85,B 0,C 180,E1 -11590.432,E2 -11590.432} C_VEL
LIN {X 0,Y 393.417,Z 431.039,A -85,B 0,C 180,E1 -11592.052,E2 -11592.052} C_VEL
LIN {X 0,Y 392.181,Z 440.418,A -85,B 0,C 180,E1 -11593.606,E2 -11593.606} C_VEL
LIN {X 0,Y 391.012,Z 449.645,A -85,B 0,C 180,E1 -11595.426,E2 -11595.426} C_VEL
LIN {X 0,Y 390.129,Z 458.329,A -85,B 0,C 180,E1 -11597.515,E2 -11597.515} C_VEL
LIN {X 0,Y 389.361,Z 465.296,A -85,B 0,C 180,E1 -11599.601,E2 -11599.601} C_VEL
LIN {X 0,Y 388.986,Z 470.773,A -85,B 0,C 180,E1 -11601.689,E2 -11601.689} C_VEL
LIN {X 0,Y 388.771,Z 475.059,A -85,B 0,C 180,E1 -11603.858,E2 -11603.858} C_VEL
LIN {X 0,Y 388.657,Z 477.814,A -85,B 0,C 180,E1 -11605.852,E2 -11605.852} C_VEL
LIN {X 0,Y 388.61,Z 479.544,A -85,B 0,C 180,E1 -11607.927,E2 -11607.927} C_VEL
LIN {X 0,Y 388.669,Z 480.137,A -85,B 0,C 180,E1 -11610,E2 -11610} C_VEL
LIN {X 0,Y 388.61,Z 479.538,A -85,B 0,C 180,E1 -11612.073,E2 -11612.073} C_VEL
LIN {X 0,Y 388.658,Z 477.801,A -85,B 0,C 180,E1 -11614.148,E2 -11614.148} C_VEL
LIN {X 0,Y 388.796,Z 474.897,A -85,B 0,C 180,E1 -11616.226,E2 -11616.226} C_VEL
LIN {X 0,Y 388.977,Z 470.757,A -85,B 0,C 180,E1 -11618.311,E2 -11618.311} C_VEL
LIN {X 0,Y 389.352,Z 465.271,A -85,B 0,C 180,E1 -11620.399,E2 -11620.399} C_VEL
LIN {X 0,Y 390.119,Z 458.29,A -85,B 0,C 180,E1 -11622.485,E2 -11622.485} C_VEL
LIN {X 0,Y 390.862,Z 450.931,A -85,B 0,C 180,E1 -11624.287,E2 -11624.287} C_VEL
LIN {X 0,Y 391.993,Z 441.808,A -85,B 0,C 180,E1 -11626.135,E2 -11626.135} C_VEL
LIN {X 0,Y 393.17,Z 432.613,A -85,B 0,C 180,E1 -11627.691,E2 -11627.691} C_VEL
LIN {X 0,Y 394.433,Z 422.081,A -85,B 0,C 180,E1 -11629.204,E2 -11629.204} C_VEL
LIN {X 0,Y 396.005,Z 409.95,A -85,B 0,C 180,E1 -11630.654,E2 -11630.654} C_VEL
LIN {X 0,Y 397.501,Z 397.013,A -85,B 0,C 180,E1 -11631.932,E2 -11631.932} C_VEL
LIN {X 0,Y 398.933,Z 384.485,A -85,B 0,C 180,E1 -11632.941,E2 -11632.941} C_VEL
LIN {X 0,Y 400.196,Z 371.018,A -85,B 0,C 180,E1 -11633.823,E2 -11633.823} C_VEL
LIN {X 0,Y 401.277,Z 356.535,A -85,B 0,C 180,E1 -11634.561,E2 -11634.561} C_VEL
LIN {X 0,Y 402.184,Z 341.671,A -85,B 0,C 180,E1 -11635.107,E2 -11635.107} C_VEL
LIN {X 0,Y 402.747,Z 325.689,A -85,B 0,C 180,E1 -11635.484,E2 -11635.484} C_VEL
LIN {X 0,Y 405.281,Z 205.183,A -85,B 0,C 180,E1 -11637.649,E2 -11637.649} C_VEL
LIN {X 0,Y 401.515,Z 185.361,A -85,B 0,C 180,E1 -11638.324,E2 -11638.324} C_VEL
LIN {X 0,Y 399.95,Z 179.198,A -85,B 0,C 180,E1 -11638.567,E2 -11638.567} C_VEL
LIN {X 0,Y 395.408,Z 168.654,A -85,B 0,C 180,E1 -11639.166,E2 -11639.166} C_VEL
LIN {X 0,Y 392.283,Z 156.024,A -85,B 0,C 180,E1 -11641.9,E2 -11641.9} C_VEL
LIN {X 0,Y 390.097,Z 147.588,A -85,B 0,C 180,E1 -11643.874,E2 -11643.874} C_VEL
LIN {X 0,Y 390.058,Z 147.513,A -85,B 0,C 180,E1 -11646.483,E2 -11646.483} C_VEL
LIN {X 0,Y 390.068,Z 147.506,A -85,B 0,C 180,E1 -11649.218,E2 -11649.218} C_VEL
LIN {X 0,Y 390.043,Z 147.52,A -85,B 0,C 180,E1 -11652.374,E2 -11652.374} C_VEL
LIN {X 0,Y 390.044,Z 147.516,A -85,B 0,C 180,E1 -11655.355,E2 -11655.355} C_VEL
LIN {X 0,Y 390.031,Z 147.511,A -85,B 0,C 180,E1 -11658.187,E2 -11658.187} C_VEL
LIN {X 0,Y 390.09,Z 147.504,A -85,B 0,C 180,E1 -11660.908,E2 -11660.908} C_VEL
LIN {X 0,Y 390.082,Z 147.504,A -85,B 0,C 180,E1 -11664.793,E2 -11664.793} C_VEL
LIN {X 0,Y 390.023,Z 147.5,A -85,B 0,C 180,E1 -11668.496,E2 -11668.496} C_VEL
LIN {X 0,Y 390.118,Z 147.512,A -85,B 0,C 180,E1 -11672.07,E2 -11672.07} C_VEL
LIN {X 0,Y 390.082,Z 147.52,A -85,B 0,C 180,E1 -11675.52,E2 -11675.52} C_VEL
LIN {X 0,Y 390.057,Z 147.511,A -85,B 0,C 180,E1 -11678.878,E2 -11678.878} C_VEL
LIN {X 0,Y 390.127,Z 147.512,A -85,B 0,C 180,E1 -11682.167,E2 -11682.167} C_VEL
LIN {X 0,Y 390.145,Z 147.504,A -85,B 0,C 180,E1 -11685.393,E2 -11685.393} C_VEL
LIN {X 0,Y 390.149,Z 147.509,A -85,B 0,C 180,E1 -11688.571,E2 -11688.571} C_VEL
LIN {X 0,Y 390.26,Z 147.49,A -85,B 0,C 180,E1 -11692.084,E2 -11692.084} C_VEL
LIN {X 0,Y 390.218,Z 147.494,A -85,B 0,C 180,E1 -11694.833,E2 -11694.833} C_VEL
LIN {X 0,Y 390.417,Z 147.468,A -85,B 0,C 180,E1 -11697.937,E2 -11697.937} C_VEL
LIN {X 0,Y 390.546,Z 147.46,A -85,B 0,C 180,E1 -11700,E2 -11700} C_VEL
LIN {X 0,Y 390.274,Z 147.483,A -85,B 0,C 180,E1 -11703.097,E2 -11703.097} C_VEL
LIN {X 0,Y 390.285,Z 147.491,A -85,B 0,C 180,E1 -11706.492,E2 -11706.492} C_VEL
LIN {X 0,Y 390.195,Z 147.493,A -85,B 0,C 180,E1 -11709.329,E2 -11709.329} C_VEL
LIN {X 0,Y 390.172,Z 147.505,A -85,B 0,C 180,E1 -11712.483,E2 -11712.483} C_VEL
LIN {X 0,Y 390.135,Z 147.503,A -85,B 0,C 180,E1 -11715.677,E2 -11715.677} C_VEL
LIN {X 0,Y 390.102,Z 147.509,A -85,B 0,C 180,E1 -11718.922,E2 -11718.922} C_VEL
LIN {X 0,Y 390.037,Z 147.526,A -85,B 0,C 180,E1 -11722.234,E2 -11722.234} C_VEL
LIN {X 0,Y 390.051,Z 147.513,A -85,B 0,C 180,E1 -11725.722,E2 -11725.722} C_VEL
LIN {X 0,Y 390.029,Z 147.522,A -85,B 0,C 180,E1 -11729.112,E2 -11729.112} C_VEL
LIN {X 0,Y 390.041,Z 147.481,A -85,B 0,C 180,E1 -11732.722,E2 -11732.722} C_VEL
LIN {X 0,Y 390.054,Z 147.525,A -85,B 0,C 180,E1 -11735.825,E2 -11735.825} C_VEL
LIN {X 0,Y 390.037,Z 147.496,A -85,B 0,C 180,E1 -11739.212,E2 -11739.212} C_VEL
LIN {X 0,Y 390.03,Z 147.521,A -85,B 0,C 180,E1 -11742.372,E2 -11742.372} C_VEL
LIN {X 0,Y 390.041,Z 147.509,A -85,B 0,C 180,E1 -11745.354,E2 -11745.354} C_VEL
LIN {X 0,Y 390.015,Z 147.528,A -85,B 0,C 180,E1 -11748.185,E2 -11748.185} C_VEL
LIN {X 0,Y 390.058,Z 147.512,A -85,B 0,C 180,E1 -11750.904,E2 -11750.904} C_VEL
LIN {X 0,Y 390.07,Z 147.521,A -85,B 0,C 180,E1 -11754.791,E2 -11754.791} C_VEL
LIN {X 0,Y 390.092,Z 147.609,A -85,B 0,C 180,E1 -11757.283,E2 -11757.283} C_VEL
LIN {X 0,Y 390.738,Z 150.358,A -85,B 0,C 180,E1 -11758.007,E2 -11758.007} C_VEL
LIN {X 0,Y 393.743,Z 162.157,A -85,B 0,C 180,E1 -11760.716,E2 -11760.716} C_VEL
LIN {X 0,Y 395.609,Z 166.408,A -85,B 0,C 180,E1 -11761.008,E2 -11761.008} C_VEL
LIN {X 0,Y 402.913,Z 183.416,A -85,B 0,C 180,E1 -11761.921,E2 -11761.921} C_VEL
LIN {X 0,Y 405.384,Z 195.286,A -85,B 0,C 180,E1 -11762.341,E2 -11762.341} C_VEL
LIN {X 0,Y 403.106,Z 307.625,A -85,B 0,C 180,E1 -11764.368,E2 -11764.368} C_VEL
LIN {X 0,Y 402.525,Z 329.953,A -85,B 0,C 180,E1 -11764.812,E2 -11764.812} C_VEL
LIN {X 0,Y 401.756,Z 344.748,A -85,B 0,C 180,E1 -11765.291,E2 -11765.291} C_VEL
LIN {X 0,Y 400.856,Z 358.737,A -85,B 0,C 180,E1 -11765.932,E2 -11765.932} C_VEL
LIN {X 0,Y 399.746,Z 371.619,A -85,B 0,C 180,E1 -11766.698,E2 -11766.698} C_VEL
LIN {X 0,Y 398.328,Z 385.227,A -85,B 0,C 180,E1 -11767.707,E2 -11767.707} C_VEL
LIN {X 0,Y 396.932,Z 397.744,A -85,B 0,C 180,E1 -11768.853,E2 -11768.853} C_VEL
LIN {X 0,Y 395.507,Z 409.358,A -85,B 0,C 180,E1 -11770.133,E2 -11770.133} C_VEL
LIN {X 0,Y 394.205,Z 420.144,A -85,B 0,C 180,E1 -11771.552,E2 -11771.552} C_VEL
LIN {X 0,Y 392.87,Z 430.119,A -85,B 0,C 180,E1 -11773.1,E2 -11773.1} C_VEL
LIN {X 0,Y 391.606,Z 439.861,A -85,B 0,C 180,E1 -11774.917,E2 -11774.917} C_VEL
LIN {X 0,Y 390.648,Z 447.982,A -85,B 0,C 180,E1 -11776.739,E2 -11776.739} C_VEL
LIN {X 0,Y 389.927,Z 454.682,A -85,B 0,C 180,E1 -11778.565,E2 -11778.565} C_VEL
LIN {X 0,Y 389.325,Z 460.89,A -85,B 0,C 180,E1 -11780.65,E2 -11780.65} C_VEL
LIN {X 0,Y 388.931,Z 465.685,A -85,B 0,C 180,E1 -11782.733,E2 -11782.733} C_VEL
LIN {X 0,Y 388.768,Z 469.199,A -85,B 0,C 180,E1 -11784.814,E2 -11784.814} C_VEL
LIN {X 0,Y 388.629,Z 471.524,A -85,B 0,C 180,E1 -11786.89,E2 -11786.89} C_VEL
LIN {X 0,Y 388.641,Z 472.447,A -85,B 0,C 180,E1 -11788.36,E2 -11788.36} C_VEL
LIN {X 0,Y 387.965,Z 472.768,A -85,B 0,C 180,E1 -11789.224,E2 -11789.224} C_VEL
LIN {X 0,Y 385.075,Z 472.824,A -85,B 0,C 180,E1 -11790.63,E2 -11790.63} C_VEL
LIN {X 0,Y 382.64,Z 472.515,A -85,B 0,C 180,E1 -11791.765,E2 -11791.765} C_VEL
LIN {X 0,Y 381.608,Z 472.064,A -85,B 0,C 180,E1 -11792.642,E2 -11792.642} C_VEL
LIN {X 0,Y 381.532,Z 471.822,A -85,B 0,C 180,E1 -11792.939,E2 -11792.939} C_VEL
LIN {X 0,Y 381.615,Z 470.683,A -85,B 0,C 180,E1 -11794.225,E2 -11794.225} C_VEL
LIN {X 0,Y 381.709,Z 467.832,A -85,B 0,C 180,E1 -11796.343,E2 -11796.343} C_VEL
LIN {X 0,Y 382.054,Z 463.749,A -85,B 0,C 180,E1 -11798.463,E2 -11798.463} C_VEL
LIN {X 0,Y 382.508,Z 458.339,A -85,B 0,C 180,E1 -11800.587,E2 -11800.587} C_VEL
LIN {X 0,Y 383.375,Z 451.444,A -85,B 0,C 180,E1 -11802.708,E2 -11802.708} C_VEL
LIN {X 0,Y 384.317,Z 442.842,A -85,B 0,C 180,E1 -11804.834,E2 -11804.834} C_VEL
LIN {X 0,Y 385.55,Z 433.697,A -85,B 0,C 180,E1 -11806.684,E2 -11806.684} C_VEL
LIN {X 0,Y 386.85,Z 424.379,A -85,B 0,C 180,E1 -11808.263,E2 -11808.263} C_VEL
LIN {X 0,Y 388.377,Z 412.892,A -85,B 0,C 180,E1 -11809.895,E2 -11809.895} C_VEL
LIN {X 0,Y 390.071,Z 400.025,A -85,B 0,C 180,E1 -11811.398,E2 -11811.398} C_VEL
LIN {X 0,Y 391.684,Z 386.451,A -85,B 0,C 180,E1 -11812.692,E2 -11812.692} C_VEL
LIN {X 0,Y 393.138,Z 373.105,A -85,B 0,C 180,E1 -11813.717,E2 -11813.717} C_VEL
LIN {X 0,Y 394.398,Z 358.611,A -85,B 0,C 180,E1 -11814.601,E2 -11814.601} C_VEL
LIN {X 0,Y 395.412,Z 344.473,A -85,B 0,C 180,E1 -11815.25,E2 -11815.25} C_VEL
LIN {X 0,Y 396.156,Z 329.908,A -85,B 0,C 180,E1 -11815.727,E2 -11815.727} C_VEL
LIN {X 0,Y 396.84,Z 303.946,A -85,B 0,C 180,E1 -11816.244,E2 -11816.244} C_VEL
LIN {X 0,Y 399.173,Z 196.671,A -85,B 0,C 180,E1 -11818.204,E2 -11818.204} C_VEL
LIN {X 0,Y 396.602,Z 185.141,A -85,B 0,C 180,E1 -11818.637,E2 -11818.637} C_VEL
LIN {X 0,Y 388.167,Z 165.978,A -85,B 0,C 180,E1 -11819.719,E2 -11819.719} C_VEL
LIN {X 0,Y 386.532,Z 162.248,A -85,B 0,C 180,E1 -11819.985,E2 -11819.985} C_VEL
LIN {X 0,Y 383.432,Z 150.067,A -85,B 0,C 180,E1 -11822.865,E2 -11822.865} C_VEL
LIN {X 0,Y 383.064,Z 148.43,A -85,B 0,C 180,E1 -11823.364,E2 -11823.364} C_VEL
LIN {X 0,Y 382.99,Z 148.397,A -85,B 0,C 180,E1 -11827.269,E2 -11827.269} C_VEL
LIN {X 0,Y 382.975,Z 148.39,A -85,B 0,C 180,E1 -11829.963,E2 -11829.963} C_VEL
LIN {X 0,Y 383.007,Z 148.394,A -85,B 0,C 180,E1 -11832.779,E2 -11832.779} C_VEL
LIN {X 0,Y 382.99,Z 148.4,A -85,B 0,C 180,E1 -11835.788,E2 -11835.788} C_VEL
LIN {X 0,Y 382.962,Z 148.381,A -85,B 0,C 180,E1 -11838.801,E2 -11838.801} C_VEL
LIN {X 0,Y 382.994,Z 148.392,A -85,B 0,C 180,E1 -11842.098,E2 -11842.098} C_VEL
LIN {X 0,Y 383.018,Z 148.391,A -85,B 0,C 180,E1 -11845.332,E2 -11845.332} C_VEL
LIN {X 0,Y 382.982,Z 148.367,A -85,B 0,C 180,E1 -11849.081,E2 -11849.081} C_VEL
LIN {X 0,Y 382.983,Z 148.404,A -85,B 0,C 180,E1 -11852.692,E2 -11852.692} C_VEL
LIN {X 0,Y 383.011,Z 148.394,A -85,B 0,C 180,E1 -11856.191,E2 -11856.191} C_VEL
LIN {X 0,Y 383.057,Z 148.383,A -85,B 0,C 180,E1 -11859.598,E2 -11859.598} C_VEL
LIN {X 0,Y 383.071,Z 148.391,A -85,B 0,C 180,E1 -11862.93,E2 -11862.93} C_VEL
LIN {X 0,Y 383.128,Z 148.376,A -85,B 0,C 180,E1 -11866.464,E2 -11866.464} C_VEL
LIN {X 0,Y 383.145,Z 148.372,A -85,B 0,C 180,E1 -11870.498,E2 -11870.498} C_VEL
LIN {X 0,Y 383.265,Z 148.366,A -85,B 0,C 180,E1 -11873.683,E2 -11873.683} C_VEL
LIN {X 0,Y 383.378,Z 148.339,A -85,B 0,C 180,E1 -11877.899,E2 -11877.899} C_VEL
LIN {X 0,Y 383.514,Z 148.336,A -85,B 0,C 180,E1 -11880,E2 -11880} C_VEL
LIN {X 0,Y 383.217,Z 148.359,A -85,B 0,C 180,E1 -11883.154,E2 -11883.154} C_VEL
LIN {X 0,Y 383.258,Z 148.366,A -85,B 0,C 180,E1 -11886.317,E2 -11886.317} C_VEL
LIN {X 0,Y 383.145,Z 148.368,A -85,B 0,C 180,E1 -11889.502,E2 -11889.502} C_VEL
LIN {X 0,Y 383.138,Z 148.385,A -85,B 0,C 180,E1 -11892.716,E2 -11892.716} C_VEL
LIN {X 0,Y 383.082,Z 148.379,A -85,B 0,C 180,E1 -11895.973,E2 -11895.973} C_VEL
LIN {X 0,Y 383.06,Z 148.39,A -85,B 0,C 180,E1 -11899.284,E2 -11899.284} C_VEL
LIN {X 0,Y 382.992,Z 148.399,A -85,B 0,C 180,E1 -11902.666,E2 -11902.666} C_VEL
LIN {X 0,Y 383.08,Z 148.378,A -85,B 0,C 180,E1 -11906.123,E2 -11906.123} C_VEL
LIN {X 0,Y 383.042,Z 148.398,A -85,B 0,C 180,E1 -11908.492,E2 -11908.492} C_VEL
LIN {X 0,Y 383.008,Z 148.36,A -85,B 0,C 180,E1 -11912.15,E2 -11912.15} C_VEL
LIN {X 0,Y 383.017,Z 148.374,A -85,B 0,C 180,E1 -11914.668,E2 -11914.668} C_VEL
LIN {X 0,Y 383,Z 148.401,A -85,B 0,C 180,E1 -11917.903,E2 -11917.903} C_VEL
LIN {X 0,Y 382.984,Z 148.381,A -85,B 0,C 180,E1 -11921.347,E2 -11921.347} C_VEL
LIN {X 0,Y 382.996,Z 148.397,A -85,B 0,C 180,E1 -11924.303,E2 -11924.303} C_VEL
LIN {X 0,Y 383.011,Z 148.389,A -85,B 0,C 180,E1 -11927.24,E2 -11927.24} C_VEL
LIN {X 0,Y 383.014,Z 148.384,A -85,B 0,C 180,E1 -11930.414,E2 -11930.414} C_VEL
LIN {X 0,Y 383.026,Z 148.387,A -85,B 0,C 180,E1 -11934.044,E2 -11934.044} C_VEL
LIN {X 0,Y 383.072,Z 148.576,A -85,B 0,C 180,E1 -11935.648,E2 -11935.648} C_VEL
LIN {X 0,Y 386.506,Z 161.636,A -85,B 0,C 180,E1 -11938.718,E2 -11938.718} C_VEL
LIN {X 0,Y 388.131,Z 168.488,A -85,B 0,C 180,E1 -11940.21,E2 -11940.21} C_VEL
LIN {X 0,Y 394.518,Z 183.173,A -85,B 0,C 180,E1 -11941.071,E2 -11941.071} C_VEL
LIN {X 0,Y 398.974,Z 205.33,A -85,B 0,C 180,E1 -11941.867,E2 -11941.867} C_VEL
LIN {X 0,Y 396.199,Z 333.843,A -85,B 0,C 180,E1 -11944.24,E2 -11944.24} C_VEL
LIN {X 0,Y 395.369,Z 349.33,A -85,B 0,C 180,E1 -11944.711,E2 -11944.711} C_VEL
LIN {X 0,Y 394.229,Z 364.632,A -85,B 0,C 180,E1 -11945.393,E2 -11945.393} C_VEL
LIN {X 0,Y 392.954,Z 379.228,A -85,B 0,C 180,E1 -11946.271,E2 -11946.271} C_VEL
LIN {X 0,Y 391.451,Z 392.694,A -85,B 0,C 180,E1 -11947.294,E2 -11947.294} C_VEL
LIN {X 0,Y 389.813,Z 406.403,A -85,B 0,C 180,E1 -11948.587,E2 -11948.587} C_VEL
LIN {X 0,Y 388.195,Z 419.001,A -85,B 0,C 180,E1 -11950.043,E2 -11950.043} C_VEL
LIN {X 0,Y 386.631,Z 430.975,A -85,B 0,C 180,E1 -11951.726,E2 -11951.726} C_VEL
LIN {X 0,Y 385.306,Z 440.353,A -85,B 0,C 180,E1 -11953.305,E2 -11953.305} C_VEL
LIN {X 0,Y 384.085,Z 449.579,A -85,B 0,C 180,E1 -11955.157,E2 -11955.157} C_VEL
LIN {X 0,Y 383.192,Z 457.253,A -85,B 0,C 180,E1 -11957.016,E2 -11957.016} C_VEL
LIN {X 0,Y 382.526,Z 463.615,A -85,B 0,C 180,E1 -11958.877,E2 -11958.877} C_VEL
LIN {X 0,Y 382.021,Z 469.462,A -85,B 0,C 180,E1 -11961.003,E2 -11961.003} C_VEL
LIN {X 0,Y 381.796,Z 472.937,A -85,B 0,C 180,E1 -11962.597,E2 -11962.597} C_VEL
LIN {X 0,Y 381.597,Z 476.447,A -85,B 0,C 180,E1 -11964.716,E2 -11964.716} C_VEL
LIN {X 0,Y 381.498,Z 478.756,A -85,B 0,C 180,E1 -11966.832,E2 -11966.832} C_VEL
LIN {X 0,Y 381.55,Z 479.917,A -85,B 0,C 180,E1 -11968.945,E2 -11968.945} C_VEL
LIN {X 0,Y 381.55,Z 479.915,A -85,B 0,C 180,E1 -11971.055,E2 -11971.055} C_VEL
LIN {X 0,Y 381.499,Z 478.745,A -85,B 0,C 180,E1 -11973.168,E2 -11973.168} C_VEL
LIN {X 0,Y 381.602,Z 476.431,A -85,B 0,C 180,E1 -11975.284,E2 -11975.284} C_VEL
LIN {X 0,Y 381.834,Z 472.92,A -85,B 0,C 180,E1 -11977.403,E2 -11977.403} C_VEL
LIN {X 0,Y 382.107,Z 468.123,A -85,B 0,C 180,E1 -11979.528,E2 -11979.528} C_VEL
LIN {X 0,Y 382.747,Z 461.911,A -85,B 0,C 180,E1 -11981.653,E2 -11981.653} C_VEL
LIN {X 0,Y 383.484,Z 454.106,A -85,B 0,C 180,E1 -11983.783,E2 -11983.783} C_VEL
LIN {X 0,Y 384.595,Z 445.806,A -85,B 0,C 180,E1 -11985.637,E2 -11985.637} C_VEL
LIN {X 0,Y 385.869,Z 435.804,A -85,B 0,C 180,E1 -11987.489,E2 -11987.489} C_VEL
LIN {X 0,Y 387.299,Z 425.573,A -85,B 0,C 180,E1 -11989.064,E2 -11989.064} C_VEL
LIN {X 0,Y 388.91,Z 413.38,A -85,B 0,C 180,E1 -11990.633,E2 -11990.633} C_VEL
LIN {X 0,Y 390.566,Z 399.799,A -85,B 0,C 180,E1 -11992.063,E2 -11992.063} C_VEL
LIN {X 0,Y 392.159,Z 386.18,A -85,B 0,C 180,E1 -11993.22,E2 -11993.22} C_VEL
LIN {X 0,Y 393.597,Z 372.069,A -85,B 0,C 180,E1 -11994.178,E2 -11994.178} C_VEL
LIN {X 0,Y 394.812,Z 356.886,A -85,B 0,C 180,E1 -11994.971,E2 -11994.971} C_VEL
LIN {X 0,Y 395.784,Z 341.592,A -85,B 0,C 180,E1 -11995.542,E2 -11995.542} C_VEL
LIN {X 0,Y 396.364,Z 325.602,A -85,B 0,C 180,E1 -11995.924,E2 -11995.924} C_VEL
LIN {X 0,Y 398.954,Z 206.17,A -85,B 0,C 180,E1 -11998.105,E2 -11998.105} C_VEL
LIN {X 0,Y 395.586,Z 188.228,A -85,B 0,C 180,E1 -11998.728,E2 -11998.728} C_VEL
LIN {X 0,Y 394.149,Z 182.274,A -85,B 0,C 180,E1 -11998.963,E2 -11998.963} C_VEL
LIN {X 0,Y 388.136,Z 168.513,A -85,B 0,C 180,E1 -11999.772,E2 -11999.772} C_VEL
LIN {X 0,Y 385.218,Z 156.69,A -85,B 0,C 180,E1 -12002.402,E2 -12002.402} C_VEL
LIN {X 0,Y 383.05,Z 148.447,A -85,B 0,C 180,E1 -12004.406,E2 -12004.406} C_VEL
LIN {X 0,Y 382.999,Z 148.402,A -85,B 0,C 180,E1 -12007.904,E2 -12007.904} C_VEL
LIN {X 0,Y 382.984,Z 148.404,A -85,B 0,C 180,E1 -12011.347,E2 -12011.347} C_VEL
LIN {X 0,Y 382.996,Z 148.383,A -85,B 0,C 180,E1 -12014.303,E2 -12014.303} C_VEL
LIN {X 0,Y 383.01,Z 148.399,A -85,B 0,C 180,E1 -12017.24,E2 -12017.24} C_VEL
LIN {X 0,Y 383.015,Z 148.377,A -85,B 0,C 180,E1 -12020.414,E2 -12020.414} C_VEL
LIN {X 0,Y 383.024,Z 148.392,A -85,B 0,C 180,E1 -12024.044,E2 -12024.044} C_VEL
LIN {X 0,Y 382.985,Z 148.361,A -85,B 0,C 180,E1 -12027.579,E2 -12027.579} C_VEL
LIN {X 0,Y 382.993,Z 148.398,A -85,B 0,C 180,E1 -12030.3,E2 -12030.3} C_VEL
LIN {X 0,Y 383.057,Z 148.392,A -85,B 0,C 180,E1 -12032.698,E2 -12032.698} C_VEL
LIN {X 0,Y 383.053,Z 148.388,A -85,B 0,C 180,E1 -12035.04,E2 -12035.04} C_VEL
LIN {X 0,Y 382.994,Z 148.392,A -85,B 0,C 180,E1 -12038.469,E2 -12038.469} C_VEL
LIN {X 0,Y 383.062,Z 148.392,A -85,B 0,C 180,E1 -12041.827,E2 -12041.827} C_VEL
LIN {X 0,Y 383.111,Z 148.376,A -85,B 0,C 180,E1 -12045.118,E2 -12045.118} C_VEL
LIN {X 0,Y 383.099,Z 148.389,A -85,B 0,C 180,E1 -12048.358,E2 -12048.358} C_VEL
LIN {X 0,Y 383.222,Z 148.367,A -85,B 0,C 180,E1 -12052.022,E2 -12052.022} C_VEL
LIN {X 0,Y 383.189,Z 148.37,A -85,B 0,C 180,E1 -12054.738,E2 -12054.738} C_VEL
LIN {X 0,Y 383.385,Z 148.344,A -85,B 0,C 180,E1 -12057.899,E2 -12057.899} C_VEL
LIN {X 0,Y 383.515,Z 148.335,A -85,B 0,C 180,E1 -12060,E2 -12060} C_VEL
LIN {X 0,Y 383.212,Z 148.362,A -85,B 0,C 180,E1 -12063.154,E2 -12063.154} C_VEL
LIN {X 0,Y 383.249,Z 148.367,A -85,B 0,C 180,E1 -12066.478,E2 -12066.478} C_VEL
LIN {X 0,Y 383.145,Z 148.372,A -85,B 0,C 180,E1 -12069.502,E2 -12069.502} C_VEL
LIN {X 0,Y 383.127,Z 148.377,A -85,B 0,C 180,E1 -12073.536,E2 -12073.536} C_VEL
LIN {X 0,Y 383.077,Z 148.391,A -85,B 0,C 180,E1 -12077.445,E2 -12077.445} C_VEL
LIN {X 0,Y 383.03,Z 148.387,A -85,B 0,C 180,E1 -12080.647,E2 -12080.647} C_VEL
LIN {X 0,Y 383.011,Z 148.396,A -85,B 0,C 180,E1 -12083.809,E2 -12083.809} C_VEL
LIN {X 0,Y 382.982,Z 148.403,A -85,B 0,C 180,E1 -12087.308,E2 -12087.308} C_VEL
LIN {X 0,Y 382.982,Z 148.369,A -85,B 0,C 180,E1 -12090.919,E2 -12090.919} C_VEL
LIN {X 0,Y 383.017,Z 148.39,A -85,B 0,C 180,E1 -12094.668,E2 -12094.668} C_VEL
LIN {X 0,Y 382.994,Z 148.393,A -85,B 0,C 180,E1 -12097.902,E2 -12097.902} C_VEL
LIN {X 0,Y 382.96,Z 148.38,A -85,B 0,C 180,E1 -12101.351,E2 -12101.351} C_VEL
LIN {X 0,Y 382.994,Z 148.4,A -85,B 0,C 180,E1 -12104.303,E2 -12104.303} C_VEL
LIN {X 0,Y 382.997,Z 148.393,A -85,B 0,C 180,E1 -12107.238,E2 -12107.238} C_VEL
LIN {X 0,Y 382.986,Z 148.389,A -85,B 0,C 180,E1 -12110.419,E2 -12110.419} C_VEL
LIN {X 0,Y 383.015,Z 148.391,A -85,B 0,C 180,E1 -12114.043,E2 -12114.043} C_VEL
LIN {X 0,Y 383.059,Z 148.502,A -85,B 0,C 180,E1 -12116.795,E2 -12116.795} C_VEL
LIN {X 0,Y 384.178,Z 153.026,A -85,B 0,C 180,E1 -12117.96,E2 -12117.96} C_VEL
LIN {X 0,Y 386.555,Z 162.412,A -85,B 0,C 180,E1 -12120.142,E2 -12120.142} C_VEL
LIN {X 0,Y 394.668,Z 180.458,A -85,B 0,C 180,E1 -12121.218,E2 -12121.218} C_VEL
LIN {X 0,Y 397.091,Z 186.681,A -85,B 0,C 180,E1 -12121.536,E2 -12121.536} C_VEL
LIN {X 0,Y 399.113,Z 196.931,A -85,B 0,C 180,E1 -12121.899,E2 -12121.899} C_VEL
LIN {X 0,Y 396.641,Z 311.292,A -85,B 0,C 180,E1 -12123.989,E2 -12123.989} C_VEL
LIN {X 0,Y 396.065,Z 331.176,A -85,B 0,C 180,E1 -12124.407,E2 -12124.407} C_VEL
LIN {X 0,Y 395.208,Z 346.62,A -85,B 0,C 180,E1 -12124.936,E2 -12124.936} C_VEL
LIN {X 0,Y 394.256,Z 360.506,A -85,B 0,C 180,E1 -12125.609,E2 -12125.609} C_VEL
LIN {X 0,Y 393.055,Z 373.581,A -85,B 0,C 180,E1 -12126.417,E2 -12126.417} C_VEL
LIN {X 0,Y 391.597,Z 386.861,A -85,B 0,C 180,E1 -12127.442,E2 -12127.442} C_VEL
LIN {X 0,Y 389.966,Z 400.36,A -85,B 0,C 180,E1 -12128.734,E2 -12128.734} C_VEL
LIN {X 0,Y 388.502,Z 411.798,A -85,B 0,C 180,E1 -12130.065,E2 -12130.065} C_VEL
LIN {X 0,Y 387.179,Z 421.992,A -85,B 0,C 180,E1 -12131.479,E2 -12131.479} C_VEL
LIN {X 0,Y 385.828,Z 431.67,A -85,B 0,C 180,E1 -12133.055,E2 -12133.055} C_VEL
LIN {X 0,Y 384.532,Z 441.157,A -85,B 0,C 180,E1 -12134.904,E2 -12134.904} C_VEL
LIN {X 0,Y 383.575,Z 449.056,A -85,B 0,C 180,E1 -12136.76,E2 -12136.76} C_VEL
LIN {X 0,Y 382.95,Z 454.751,A -85,B 0,C 180,E1 -12138.353,E2 -12138.353} C_VEL
LIN {X 0,Y 382.297,Z 460.958,A -85,B 0,C 180,E1 -12140.477,E2 -12140.477} C_VEL
LIN {X 0,Y 381.859,Z 465.753,A -85,B 0,C 180,E1 -12142.598,E2 -12142.598} C_VEL
LIN {X 0,Y 381.673,Z 469.266,A -85,B 0,C 180,E1 -12144.717,E2 -12144.717} C_VEL
LIN {X 0,Y 381.541,Z 471.591,A -85,B 0,C 180,E1 -12146.832,E2 -12146.832} C_VEL
LIN {X 0,Y 381.557,Z 472.778,A -85,B 0,C 180,E1 -12148.945,E2 -12148.945} C_VEL
LIN {X 0,Y 381.557,Z 472.794,A -85,B 0,C 180,E1 -12151.055,E2 -12151.055} C_VEL
LIN {X 0,Y 381.532,Z 471.822,A -85,B 0,C 180,E1 -12152.939,E2 -12152.939} C_VEL
LIN {X 0,Y 380.882,Z 471.144,A -85,B 0,C 180,E1 -12153.814,E2 -12153.814} C_VEL
LIN {X 0,Y 378.057,Z 469.579,A -85,B 0,C 180,E1 -12155.23,E2 -12155.23} C_VEL
LIN {X 0,Y 375.722,Z 468.017,A -85,B 0,C 180,E1 -12156.365,E2 -12156.365} C_VEL
LIN {X 0,Y 374.812,Z 466.61,A -85,B 0,C 180,E1 -12157.236,E2 -12157.236} C_VEL
LIN {X 0,Y 374.788,Z 466.039,A -85,B 0,C 180,E1 -12157.529,E2 -12157.529} C_VEL
LIN {X 0,Y 375.22,Z 461.284,A -85,B 0,C 180,E1 -12159.705,E2 -12159.705} C_VEL
LIN {X 0,Y 375.949,Z 455.154,A -85,B 0,C 180,E1 -12161.867,E2 -12161.867} C_VEL
LIN {X 0,Y 376.829,Z 447.439,A -85,B 0,C 180,E1 -12164.032,E2 -12164.032} C_VEL
LIN {X 0,Y 377.95,Z 439.213,A -85,B 0,C 180,E1 -12165.919,E2 -12165.919} C_VEL
LIN {X 0,Y 379.355,Z 429.307,A -85,B 0,C 180,E1 -12167.799,E2 -12167.799} C_VEL
LIN {X 0,Y 381.045,Z 418.026,A -85,B 0,C 180,E1 -12169.563,E2 -12169.563} C_VEL
LIN {X 0,Y 382.64,Z 405.955,A -85,B 0,C 180,E1 -12171.128,E2 -12171.128} C_VEL
LIN {X 0,Y 384.268,Z 393.646,A -85,B 0,C 180,E1 -12172.445,E2 -12172.445} C_VEL
LIN {X 0,Y 385.87,Z 380.193,A -85,B 0,C 180,E1 -12173.622,E2 -12173.622} C_VEL
LIN {X 0,Y 387.417,Z 365.203,A -85,B 0,C 180,E1 -12174.66,E2 -12174.66} C_VEL
LIN {X 0,Y 388.572,Z 350.24,A -85,B 0,C 180,E1 -12175.458,E2 -12175.458} C_VEL
LIN {X 0,Y 389.522,Z 335.616,A -85,B 0,C 180,E1 -12176.019,E2 -12176.019} C_VEL
LIN {X 0,Y 390.128,Z 320.081,A -85,B 0,C 180,E1 -12176.407,E2 -12176.407} C_VEL
LIN {X 0,Y 392.925,Z 198.131,A -85,B 0,C 180,E1 -12178.665,E2 -12178.665} C_VEL
LIN {X 0,Y 390.786,Z 188.191,A -85,B 0,C 180,E1 -12179.042,E2 -12179.042} C_VEL
LIN {X 0,Y 383.264,Z 170.907,A -85,B 0,C 180,E1 -12180.035,E2 -12180.035} C_VEL
LIN {X 0,Y 379.356,Z 162.436,A -85,B 0,C 180,E1 -12180.598,E2 -12180.598} C_VEL
LIN {X 0,Y 376.053,Z 149.719,A -85,B 0,C 180,E1 -12183.698,E2 -12183.698} C_VEL
LIN {X 0,Y 375.985,Z 149.292,A -85,B 0,C 180,E1 -12183.947,E2 -12183.947} C_VEL
LIN {X 0,Y 375.948,Z 149.27,A -85,B 0,C 180,E1 -12186.742,E2 -12186.742} C_VEL
LIN {X 0,Y 375.939,Z 149.266,A -85,B 0,C 180,E1 -12189.961,E2 -12189.961} C_VEL
LIN {X 0,Y 375.925,Z 149.265,A -85,B 0,C 180,E1 -12193.767,E2 -12193.767} C_VEL
LIN {X 0,Y 375.934,Z 149.284,A -85,B 0,C 180,E1 -12196.811,E2 -12196.811} C_VEL
LIN {X 0,Y 375.935,Z 149.246,A -85,B 0,C 180,E1 -12200.534,E2 -12200.534} C_VEL
LIN {X 0,Y 375.963,Z 149.278,A -85,B 0,C 180,E1 -12203.496,E2 -12203.496} C_VEL
LIN {X 0,Y 375.96,Z 149.256,A -85,B 0,C 180,E1 -12205.888,E2 -12205.888} C_VEL
LIN {X 0,Y 375.962,Z 149.253,A -85,B 0,C 180,E1 -12209.687,E2 -12209.687} C_VEL
LIN {X 0,Y 375.927,Z 149.283,A -85,B 0,C 180,E1 -12212.136,E2 -12212.136} C_VEL
LIN {X 0,Y 375.937,Z 149.269,A -85,B 0,C 180,E1 -12214.534,E2 -12214.534} C_VEL
LIN {X 0,Y 375.975,Z 149.275,A -85,B 0,C 180,E1 -12216.887,E2 -12216.887} C_VEL
LIN {X 0,Y 375.996,Z 149.261,A -85,B 0,C 180,E1 -12220.339,E2 -12220.339} C_VEL
LIN {X 0,Y 375.978,Z 149.275,A -85,B 0,C 180,E1 -12223.716,E2 -12223.716} C_VEL
LIN {X 0,Y 376.106,Z 149.254,A -85,B 0,C 180,E1 -12227.042,E2 -12227.042} C_VEL
LIN {X 0,Y 376.115,Z 149.249,A -85,B 0,C 180,E1 -12230.318,E2 -12230.318} C_VEL
LIN {X 0,Y 376.222,Z 149.242,A -85,B 0,C 180,E1 -12233.564,E2 -12233.564} C_VEL
LIN {X 0,Y 376.343,Z 149.214,A -85,B 0,C 180,E1 -12237.859,E2 -12237.859} C_VEL
LIN {X 0,Y 376.483,Z 149.212,A -85,B 0,C 180,E1 -12240,E2 -12240} C_VEL
LIN {X 0,Y 376.347,Z 149.22,A -85,B 0,C 180,E1 -12242.14,E2 -12242.14} C_VEL
LIN {X 0,Y 376.216,Z 149.243,A -85,B 0,C 180,E1 -12246.435,E2 -12246.435} C_VEL
LIN {X 0,Y 376.115,Z 149.243,A -85,B 0,C 180,E1 -12249.681,E2 -12249.681} C_VEL
LIN {X 0,Y 376.091,Z 149.258,A -85,B 0,C 180,E1 -12253.657,E2 -12253.657} C_VEL
LIN {X 0,Y 376.044,Z 149.268,A -85,B 0,C 180,E1 -12257.606,E2 -12257.606} C_VEL
LIN {X 0,Y 375.98,Z 149.263,A -85,B 0,C 180,E1 -12260.832,E2 -12260.832} C_VEL
LIN {X 0,Y 375.988,Z 149.275,A -85,B 0,C 180,E1 -12264.282,E2 -12264.282} C_VEL
LIN {X 0,Y 376.02,Z 149.26,A -85,B 0,C 180,E1 -12266.652,E2 -12266.652} C_VEL
LIN {X 0,Y 375.972,Z 149.275,A -85,B 0,C 180,E1 -12269.079,E2 -12269.079} C_VEL
LIN {X 0,Y 375.948,Z 149.234,A -85,B 0,C 180,E1 -12272.828,E2 -12272.828} C_VEL
LIN {X 0,Y 375.957,Z 149.268,A -85,B 0,C 180,E1 -12275.415,E2 -12275.415} C_VEL
LIN {X 0,Y 375.974,Z 149.269,A -85,B 0,C 180,E1 -12278.27,E2 -12278.27} C_VEL
LIN {X 0,Y 375.934,Z 149.262,A -85,B 0,C 180,E1 -12281.6,E2 -12281.6} C_VEL
LIN {X 0,Y 375.927,Z 149.266,A -85,B 0,C 180,E1 -12285.268,E2 -12285.268} C_VEL
LIN {X 0,Y 375.935,Z 149.284,A -85,B 0,C 180,E1 -12288.399,E2 -12288.399} C_VEL
LIN {X 0,Y 375.974,Z 149.272,A -85,B 0,C 180,E1 -12291.729,E2 -12291.729} C_VEL
LIN {X 0,Y 375.991,Z 149.444,A -85,B 0,C 180,E1 -12295.112,E2 -12295.112} C_VEL
LIN {X 0,Y 379.208,Z 161.551,A -85,B 0,C 180,E1 -12298.043,E2 -12298.043} C_VEL
LIN {X 0,Y 380.919,Z 168.537,A -85,B 0,C 180,E1 -12299.598,E2 -12299.598} C_VEL
LIN {X 0,Y 387.565,Z 183.411,A -85,B 0,C 180,E1 -12300.507,E2 -12300.507} C_VEL
LIN {X 0,Y 388.938,Z 187.403,A -85,B 0,C 180,E1 -12300.704,E2 -12300.704} C_VEL
LIN {X 0,Y 392.665,Z 206.315,A -85,B 0,C 180,E1 -12301.395,E2 -12301.395} C_VEL
LIN {X 0,Y 390.393,Z 310.064,A -85,B 0,C 180,E1 -12303.325,E2 -12303.325} C_VEL
LIN {X 0,Y 389.685,Z 336.211,A -85,B 0,C 180,E1 -12303.849,E2 -12303.849} C_VEL
LIN {X 0,Y 388.765,Z 351.555,A -85,B 0,C 180,E1 -12304.354,E2 -12304.354} C_VEL
LIN {X 0,Y 387.704,Z 365.503,A -85,B 0,C 180,E1 -12305.007,E2 -12305.007} C_VEL
LIN {X 0,Y 386.439,Z 379.167,A -85,B 0,C 180,E1 -12305.845,E2 -12305.845} C_VEL
LIN {X 0,Y 384.903,Z 392.632,A -85,B 0,C 180,E1 -12306.885,E2 -12306.885} C_VEL
LIN {X 0,Y 383.376,Z 405.049,A -85,B 0,C 180,E1 -12308.067,E2 -12308.067} C_VEL
LIN {X 0,Y 381.768,Z 416.605,A -85,B 0,C 180,E1 -12309.386,E2 -12309.386} C_VEL
LIN {X 0,Y 380.314,Z 427.362,A -85,B 0,C 180,E1 -12310.852,E2 -12310.852} C_VEL
LIN {X 0,Y 378.821,Z 437.312,A -85,B 0,C 180,E1 -12312.454,E2 -12312.454} C_VEL
LIN {X 0,Y 377.518,Z 447.047,A -85,B 0,C 180,E1 -12314.339,E2 -12314.339} C_VEL
LIN {X 0,Y 376.496,Z 454.631,A -85,B 0,C 180,E1 -12316.09,E2 -12316.09} C_VEL
LIN {X 0,Y 375.744,Z 461.88,A -85,B 0,C 180,E1 -12318.127,E2 -12318.127} C_VEL
LIN {X 0,Y 375.06,Z 468.078,A -85,B 0,C 180,E1 -12320.291,E2 -12320.291} C_VEL
LIN {X 0,Y 374.711,Z 472.871,A -85,B 0,C 180,E1 -12322.456,E2 -12322.456} C_VEL
LIN {X 0,Y 374.514,Z 476.381,A -85,B 0,C 180,E1 -12324.616,E2 -12324.616} C_VEL
LIN {X 0,Y 374.415,Z 478.69,A -85,B 0,C 180,E1 -12326.772,E2 -12326.772} C_VEL
LIN {X 0,Y 374.448,Z 479.851,A -85,B 0,C 180,E1 -12328.925,E2 -12328.925} C_VEL
LIN {X 0,Y 374.448,Z 479.849,A -85,B 0,C 180,E1 -12331.075,E2 -12331.075} C_VEL
LIN {X 0,Y 374.416,Z 478.679,A -85,B 0,C 180,E1 -12333.228,E2 -12333.228} C_VEL
LIN {X 0,Y 374.518,Z 476.364,A -85,B 0,C 180,E1 -12335.384,E2 -12335.384} C_VEL
LIN {X 0,Y 374.74,Z 472.853,A -85,B 0,C 180,E1 -12337.544,E2 -12337.544} C_VEL
LIN {X 0,Y 375.057,Z 468.055,A -85,B 0,C 180,E1 -12339.709,E2 -12339.709} C_VEL
LIN {X 0,Y 375.738,Z 461.842,A -85,B 0,C 180,E1 -12341.873,E2 -12341.873} C_VEL
LIN {X 0,Y 376.546,Z 454.037,A -85,B 0,C 180,E1 -12344.042,E2 -12344.042} C_VEL
LIN {X 0,Y 377.699,Z 445.737,A -85,B 0,C 180,E1 -12345.93,E2 -12345.93} C_VEL
LIN {X 0,Y 379.065,Z 435.735,A -85,B 0,C 180,E1 -12347.813,E2 -12347.813} C_VEL
LIN {X 0,Y 380.52,Z 425.504,A -85,B 0,C 180,E1 -12349.418,E2 -12349.418} C_VEL
LIN {X 0,Y 382.242,Z 413.31,A -85,B 0,C 180,E1 -12351.01,E2 -12351.01} C_VEL
LIN {X 0,Y 383.945,Z 399.729,A -85,B 0,C 180,E1 -12352.464,E2 -12352.464} C_VEL
LIN {X 0,Y 385.629,Z 386.109,A -85,B 0,C 180,E1 -12353.637,E2 -12353.637} C_VEL
LIN {X 0,Y 387.126,Z 371.996,A -85,B 0,C 180,E1 -12354.608,E2 -12354.608} C_VEL
LIN {X 0,Y 388.387,Z 356.505,A -85,B 0,C 180,E1 -12355.427,E2 -12355.427} C_VEL
LIN {X 0,Y 389.387,Z 341.513,A -85,B 0,C 180,E1 -12355.992,E2 -12355.992} C_VEL
LIN {X 0,Y 390.008,Z 325.516,A -85,B 0,C 180,E1 -12356.379,E2 -12356.379} C_VEL
LIN {X 0,Y 392.677,Z 206.522,A -85,B 0,C 180,E1 -12358.586,E2 -12358.586} C_VEL
LIN {X 0,Y 388.431,Z 185.477,A -85,B 0,C 180,E1 -12359.363,E2 -12359.363} C_VEL
LIN {X 0,Y 380.941,Z 168.529,A -85,B 0,C 180,E1 -12360.384,E2 -12360.384} C_VEL
LIN {X 0,Y 377.857,Z 156.315,A -85,B 0,C 180,E1 -12363.177,E2 -12363.177} C_VEL
LIN {X 0,Y 376,Z 149.329,A -85,B 0,C 180,E1 -12364.94,E2 -12364.94} C_VEL
LIN {X 0,Y 375.973,Z 149.27,A -85,B 0,C 180,E1 -12368.27,E2 -12368.27} C_VEL
LIN {X 0,Y 375.935,Z 149.285,A -85,B 0,C 180,E1 -12371.601,E2 -12371.601} C_VEL
LIN {X 0,Y 375.927,Z 149.274,A -85,B 0,C 180,E1 -12375.269,E2 -12375.269} C_VEL
LIN {X 0,Y 375.934,Z 149.261,A -85,B 0,C 180,E1 -12378.399,E2 -12378.399} C_VEL
LIN {X 0,Y 375.974,Z 149.27,A -85,B 0,C 180,E1 -12381.73,E2 -12381.73} C_VEL
LIN {X 0,Y 375.979,Z 149.248,A -85,B 0,C 180,E1 -12385.333,E2 -12385.333} C_VEL
LIN {X 0,Y 375.957,Z 149.247,A -85,B 0,C 180,E1 -12388.438,E2 -12388.438} C_VEL
LIN {X 0,Y 375.997,Z 149.271,A -85,B 0,C 180,E1 -12392.142,E2 -12392.142} C_VEL
LIN {X 0,Y 376.007,Z 149.261,A -85,B 0,C 180,E1 -12394.539,E2 -12394.539} C_VEL
LIN {X 0,Y 375.964,Z 149.269,A -85,B 0,C 180,E1 -12398.046,E2 -12398.046} C_VEL
LIN {X 0,Y 376.008,Z 149.273,A -85,B 0,C 180,E1 -12401.473,E2 -12401.473} C_VEL
LIN {X 0,Y 376.059,Z 149.252,A -85,B 0,C 180,E1 -12404.833,E2 -12404.833} C_VEL
LIN {X 0,Y 376.051,Z 149.266,A -85,B 0,C 180,E1 -12408.137,E2 -12408.137} C_VEL
LIN {X 0,Y 376.174,Z 149.244,A -85,B 0,C 180,E1 -12411.968,E2 -12411.968} C_VEL
LIN {X 0,Y 376.16,Z 149.246,A -85,B 0,C 180,E1 -12414.64,E2 -12414.64} C_VEL
LIN {X 0,Y 376.351,Z 149.22,A -85,B 0,C 180,E1 -12417.86,E2 -12417.86} C_VEL
LIN {X 0,Y 376.485,Z 149.211,A -85,B 0,C 180,E1 -12420,E2 -12420} C_VEL
LIN {X 0,Y 376.345,Z 149.214,A -85,B 0,C 180,E1 -12422.141,E2 -12422.141} C_VEL
LIN {X 0,Y 376.218,Z 149.243,A -85,B 0,C 180,E1 -12426.461,E2 -12426.461} C_VEL
LIN {X 0,Y 376.115,Z 149.248,A -85,B 0,C 180,E1 -12429.682,E2 -12429.682} C_VEL
LIN {X 0,Y 376.091,Z 149.252,A -85,B 0,C 180,E1 -12433.658,E2 -12433.658} C_VEL
LIN {X 0,Y 376.028,Z 149.27,A -85,B 0,C 180,E1 -12437.599,E2 -12437.599} C_VEL
LIN {X 0,Y 375.98,Z 149.267,A -85,B 0,C 180,E1 -12440.832,E2 -12440.832} C_VEL
LIN {X 0,Y 375.937,Z 149.271,A -85,B 0,C 180,E1 -12444.286,E2 -12444.286} C_VEL
LIN {X 0,Y 375.921,Z 149.28,A -85,B 0,C 180,E1 -12446.66,E2 -12446.66} C_VEL
LIN {X 0,Y 375.917,Z 149.279,A -85,B 0,C 180,E1 -12449.084,E2 -12449.084} C_VEL
LIN {X 0,Y 375.939,Z 149.236,A -85,B 0,C 180,E1 -12451.564,E2 -12451.564} C_VEL
LIN {X 0,Y 375.957,Z 149.274,A -85,B 0,C 180,E1 -12455.416,E2 -12455.416} C_VEL
LIN {X 0,Y 375.937,Z 149.269,A -85,B 0,C 180,E1 -12458.263,E2 -12458.263} C_VEL
LIN {X 0,Y 375.917,Z 149.261,A -85,B 0,C 180,E1 -12461.598,E2 -12461.598} C_VEL
LIN {X 0,Y 375.924,Z 149.275,A -85,B 0,C 180,E1 -12464.731,E2 -12464.731} C_VEL
LIN {X 0,Y 375.917,Z 149.283,A -85,B 0,C 180,E1 -12467.698,E2 -12467.698} C_VEL
LIN {X 0,Y 375.935,Z 149.267,A -85,B 0,C 180,E1 -12470.534,E2 -12470.534} C_VEL
LIN {X 0,Y 375.959,Z 149.268,A -85,B 0,C 180,E1 -12473.497,E2 -12473.497} C_VEL
LIN {X 0,Y 376.005,Z 149.425,A -85,B 0,C 180,E1 -12476.297,E2 -12476.297} C_VEL
LIN {X 0,Y 379.145,Z 161.641,A -85,B 0,C 180,E1 -12479.35,E2 -12479.35} C_VEL
LIN {X 0,Y 379.55,Z 162.97,A -85,B 0,C 180,E1 -12479.564,E2 -12479.564} C_VEL
LIN {X 0,Y 388.67,Z 182.969,A -85,B 0,C 180,E1 -12480.781,E2 -12480.781} C_VEL
LIN {X 0,Y 391.12,Z 189.252,A -85,B 0,C 180,E1 -12481.112,E2 -12481.112} C_VEL
LIN {X 0,Y 392.846,Z 198.686,A -85,B 0,C 180,E1 -12481.444,E2 -12481.444} C_VEL
LIN {X 0,Y 390.295,Z 311.384,A -85,B 0,C 180,E1 -12483.534,E2 -12483.534} C_VEL
LIN {X 0,Y 389.688,Z 331.258,A -85,B 0,C 180,E1 -12483.957,E2 -12483.957} C_VEL
LIN {X 0,Y 388.773,Z 346.977,A -85,B 0,C 180,E1 -12484.505,E2 -12484.505} C_VEL
LIN {X 0,Y 387.73,Z 361.391,A -85,B 0,C 180,E1 -12485.222,E2 -12485.222} C_VEL
LIN {X 0,Y 386.357,Z 375.417,A -85,B 0,C 180,E1 -12486.125,E2 -12486.125} C_VEL
LIN {X 0,Y 384.857,Z 388.366,A -85,B 0,C 180,E1 -12487.167,E2 -12487.167} C_VEL
LIN {X 0,Y 383.186,Z 401.603,A -85,B 0,C 180,E1 -12488.48,E2 -12488.48} C_VEL
LIN {X 0,Y 381.572,Z 413.687,A -85,B 0,C 180,E1 -12489.942,E2 -12489.942} C_VEL
LIN {X 0,Y 380.139,Z 423.836,A -85,B 0,C 180,E1 -12491.403,E2 -12491.403} C_VEL
LIN {X 0,Y 378.577,Z 434.677,A -85,B 0,C 180,E1 -12493.277,E2 -12493.277} C_VEL
LIN {X 0,Y 377.294,Z 443.793,A -85,B 0,C 180,E1 -12495.187,E2 -12495.187} C_VEL
LIN {X 0,Y 376.478,Z 451.133,A -85,B 0,C 180,E1 -12497.055,E2 -12497.055} C_VEL
LIN {X 0,Y 375.51,Z 458.109,A -85,B 0,C 180,E1 -12499.213,E2 -12499.213} C_VEL
LIN {X 0,Y 375.005,Z 463.591,A -85,B 0,C 180,E1 -12501.377,E2 -12501.377} C_VEL
LIN {X 0,Y 374.689,Z 468.132,A -85,B 0,C 180,E1 -12503.783,E2 -12503.783} C_VEL
LIN {X 0,Y 374.548,Z 470.64,A -85,B 0,C 180,E1 -12505.696,E2 -12505.696} C_VEL
LIN {X 0,Y 374.452,Z 472.391,A -85,B 0,C 180,E1 -12507.849,E2 -12507.849} C_VEL
LIN {X 0,Y 374.472,Z 473.003,A -85,B 0,C 180,E1 -12510,E2 -12510} C_VEL
LIN {X 0,Y 374.452,Z 472.438,A -85,B 0,C 180,E1 -12512.151,E2 -12512.151} C_VEL
LIN {X 0,Y 374.543,Z 470.749,A -85,B 0,C 180,E1 -12514.305,E2 -12514.305} C_VEL
LIN {X 0,Y 374.628,Z 467.898,A -85,B 0,C 180,E1 -12516.463,E2 -12516.463} C_VEL
LIN {X 0,Y 374.788,Z 466.039,A -85,B 0,C 180,E1 -12517.529,E2 -12517.529} C_VEL
LIN {X 0,Y 374.293,Z 464.422,A -85,B 0,C 180,E1 -12518.394,E2 -12518.394} C_VEL
LIN {X 0,Y 371.708,Z 461.389,A -85,B 0,C 180,E1 -12519.79,E2 -12519.79} C_VEL
LIN {X 0,Y 369.235,Z 457.884,A -85,B 0,C 180,E1 -12521.177,E2 -12521.177} C_VEL
LIN {X 0,Y 368.933,Z 455.452,A -85,B 0,C 180,E1 -12522.017,E2 -12522.017} C_VEL
LIN {X 0,Y 369.846,Z 447.618,A -85,B 0,C 180,E1 -12524.273,E2 -12524.273} C_VEL
LIN {X 0,Y 371.096,Z 439.278,A -85,B 0,C 180,E1 -12526.221,E2 -12526.221} C_VEL
LIN {X 0,Y 372.549,Z 429.371,A -85,B 0,C 180,E1 -12528.136,E2 -12528.136} C_VEL
LIN {X 0,Y 374.143,Z 419.215,A -85,B 0,C 180,E1 -12529.762,E2 -12529.762} C_VEL
LIN {X 0,Y 375.693,Z 408.193,A -85,B 0,C 180,E1 -12531.25,E2 -12531.25} C_VEL
LIN {X 0,Y 377.342,Z 396.294,A -85,B 0,C 180,E1 -12532.591,E2 -12532.591} C_VEL
LIN {X 0,Y 378.949,Z 383.416,A -85,B 0,C 180,E1 -12533.79,E2 -12533.79} C_VEL
LIN {X 0,Y 380.538,Z 369.29,A -85,B 0,C 180,E1 -12534.845,E2 -12534.845} C_VEL
LIN {X 0,Y 381.825,Z 354.653,A -85,B 0,C 180,E1 -12535.7,E2 -12535.7} C_VEL
LIN {X 0,Y 382.91,Z 339.351,A -85,B 0,C 180,E1 -12536.356,E2 -12536.356} C_VEL
LIN {X 0,Y 383.625,Z 324.672,A -85,B 0,C 180,E1 -12536.78,E2 -12536.78} C_VEL
LIN {X 0,Y 386.314,Z 214.792,A -85,B 0,C 180,E1 -12538.856,E2 -12538.856} C_VEL
LIN {X 0,Y 386.59,Z 198.672,A -85,B 0,C 180,E1 -12539.169,E2 -12539.169} C_VEL
LIN {X 0,Y 384.828,Z 190.745,A -85,B 0,C 180,E1 -12539.482,E2 -12539.482} C_VEL
LIN {X 0,Y 377.083,Z 173.05,A -85,B 0,C 180,E1 -12540.534,E2 -12540.534} C_VEL
LIN {X 0,Y 372.183,Z 162.612,A -85,B 0,C 180,E1 -12541.242,E2 -12541.242} C_VEL
LIN {X 0,Y 369.453,Z 152.233,A -85,B 0,C 180,E1 -12543.808,E2 -12543.808} C_VEL
LIN {X 0,Y 368.947,Z 150.21,A -85,B 0,C 180,E1 -12544.417,E2 -12544.417} C_VEL
LIN {X 0,Y 368.896,Z 150.156,A -85,B 0,C 180,E1 -12547.564,E2 -12547.564} C_VEL
LIN {X 0,Y 368.884,Z 150.146,A -85,B 0,C 180,E1 -12550.374,E2 -12550.374} C_VEL
LIN {X 0,Y 368.878,Z 150.143,A -85,B 0,C 180,E1 -12553.615,E2 -12553.615} C_VEL
LIN {X 0,Y 368.884,Z 150.163,A -85,B 0,C 180,E1 -12556.695,E2 -12556.695} C_VEL
LIN {X 0,Y 368.885,Z 150.122,A -85,B 0,C 180,E1 -12559.648,E2 -12559.648} C_VEL
LIN {X 0,Y 368.9,Z 150.16,A -85,B 0,C 180,E1 -12563.145,E2 -12563.145} C_VEL
LIN {X 0,Y 368.897,Z 150.124,A -85,B 0,C 180,E1 -12566.462,E2 -12566.462} C_VEL
LIN {X 0,Y 368.897,Z 150.118,A -85,B 0,C 180,E1 -12569.043,E2 -12569.043} C_VEL
LIN {X 0,Y 368.912,Z 150.153,A -85,B 0,C 180,E1 -12571.558,E2 -12571.558} C_VEL
LIN {X 0,Y 368.888,Z 150.146,A -85,B 0,C 180,E1 -12575.219,E2 -12575.219} C_VEL
LIN {X 0,Y 368.921,Z 150.155,A -85,B 0,C 180,E1 -12577.604,E2 -12577.604} C_VEL
LIN {X 0,Y 368.953,Z 150.143,A -85,B 0,C 180,E1 -12581.105,E2 -12581.105} C_VEL
LIN {X 0,Y 368.957,Z 150.14,A -85,B 0,C 180,E1 -12584.533,E2 -12584.533} C_VEL
LIN {X 0,Y 369.06,Z 150.131,A -85,B 0,C 180,E1 -12586.79,E2 -12586.79} C_VEL
LIN {X 0,Y 369.065,Z 150.128,A -85,B 0,C 180,E1 -12590.132,E2 -12590.132} C_VEL
LIN {X 0,Y 369.18,Z 150.118,A -85,B 0,C 180,E1 -12593.441,E2 -12593.441} C_VEL
LIN {X 0,Y 369.307,Z 150.09,A -85,B 0,C 180,E1 -12597.819,E2 -12597.819} C_VEL
LIN {X 0,Y 369.432,Z 150.09,A -85,B 0,C 180,E1 -12600,E2 -12600} C_VEL
LIN {X 0,Y 369.311,Z 150.096,A -85,B 0,C 180,E1 -12602.181,E2 -12602.181} C_VEL
LIN {X 0,Y 369.176,Z 150.121,A -85,B 0,C 180,E1 -12606.559,E2 -12606.559} C_VEL
LIN {X 0,Y 369.065,Z 150.121,A -85,B 0,C 180,E1 -12609.868,E2 -12609.868} C_VEL
LIN {X 0,Y 369.039,Z 150.135,A -85,B 0,C 180,E1 -12613.772,E2 -12613.772} C_VEL
LIN {X 0,Y 369.003,Z 150.144,A -85,B 0,C 180,E1 -12617.768,E2 -12617.768} C_VEL
LIN {X 0,Y 368.911,Z 150.144,A -85,B 0,C 180,E1 -12621.221,E2 -12621.221} C_VEL
LIN {X 0,Y 368.955,Z 150.146,A -85,B 0,C 180,E1 -12624.775,E2 -12624.775} C_VEL
LIN {X 0,Y 368.969,Z 150.144,A -85,B 0,C 180,E1 -12627.203,E2 -12627.203} C_VEL
LIN {X 0,Y 368.92,Z 150.151,A -85,B 0,C 180,E1 -12629.69,E2 -12629.69} C_VEL
LIN {X 0,Y 368.896,Z 150.111,A -85,B 0,C 180,E1 -12633.043,E2 -12633.043} C_VEL
LIN {X 0,Y 368.917,Z 150.152,A -85,B 0,C 180,E1 -12636.197,E2 -12636.197} C_VEL
LIN {X 0,Y 368.903,Z 150.141,A -85,B 0,C 180,E1 -12638.953,E2 -12638.953} C_VEL
LIN {X 0,Y 368.882,Z 150.148,A -85,B 0,C 180,E1 -12642.009,E2 -12642.009} C_VEL
LIN {X 0,Y 368.88,Z 150.144,A -85,B 0,C 180,E1 -12645.176,E2 -12645.176} C_VEL
LIN {X 0,Y 368.884,Z 150.161,A -85,B 0,C 180,E1 -12648.177,E2 -12648.177} C_VEL
LIN {X 0,Y 368.908,Z 150.146,A -85,B 0,C 180,E1 -12651.36,E2 -12651.36} C_VEL
LIN {X 0,Y 368.975,Z 150.379,A -85,B 0,C 180,E1 -12654.576,E2 -12654.576} C_VEL
LIN {X 0,Y 372.04,Z 161.826,A -85,B 0,C 180,E1 -12657.427,E2 -12657.427} C_VEL
LIN {X 0,Y 373.654,Z 168.433,A -85,B 0,C 180,E1 -12658.94,E2 -12658.94} C_VEL
LIN {X 0,Y 380.864,Z 184.371,A -85,B 0,C 180,E1 -12659.957,E2 -12659.957} C_VEL
LIN {X 0,Y 383.007,Z 189.81,A -85,B 0,C 180,E1 -12660.257,E2 -12660.257} C_VEL
LIN {X 0,Y 386.426,Z 207.619,A -85,B 0,C 180,E1 -12660.917,E2 -12660.917} C_VEL
LIN {X 0,Y 384.07,Z 310.018,A -85,B 0,C 180,E1 -12662.85,E2 -12662.85} C_VEL
LIN {X 0,Y 383.344,Z 336.157,A -85,B 0,C 180,E1 -12663.383,E2 -12663.383} C_VEL
LIN {X 0,Y 382.361,Z 351.743,A -85,B 0,C 180,E1 -12663.904,E2 -12663.904} C_VEL
LIN {X 0,Y 381.199,Z 366.322,A -85,B 0,C 180,E1 -12664.607,E2 -12664.607} C_VEL
LIN {X 0,Y 379.743,Z 380.909,A -85,B 0,C 180,E1 -12665.537,E2 -12665.537} C_VEL
LIN {X 0,Y 378.162,Z 394.079,A -85,B 0,C 180,E1 -12666.594,E2 -12666.594} C_VEL
LIN {X 0,Y 376.408,Z 407.488,A -85,B 0,C 180,E1 -12667.929,E2 -12667.929} C_VEL
LIN {X 0,Y 374.777,Z 418.768,A -85,B 0,C 180,E1 -12669.282,E2 -12669.282} C_VEL
LIN {X 0,Y 373.076,Z 430.846,A -85,B 0,C 180,E1 -12671.037,E2 -12671.037} C_VEL
LIN {X 0,Y 371.596,Z 440.223,A -85,B 0,C 180,E1 -12672.67,E2 -12672.67} C_VEL
LIN {X 0,Y 370.252,Z 449.449,A -85,B 0,C 180,E1 -12674.589,E2 -12674.589} C_VEL
LIN {X 0,Y 369.126,Z 458.132,A -85,B 0,C 180,E1 -12676.793,E2 -12676.793} C_VEL
LIN {X 0,Y 368.518,Z 463.483,A -85,B 0,C 180,E1 -12678.449,E2 -12678.449} C_VEL
LIN {X 0,Y 367.895,Z 469.33,A -85,B 0,C 180,E1 -12680.655,E2 -12680.655} C_VEL
LIN {X 0,Y 367.65,Z 472.805,A -85,B 0,C 180,E1 -12682.31,E2 -12682.31} C_VEL
LIN {X 0,Y 367.436,Z 476.315,A -85,B 0,C 180,E1 -12684.512,E2 -12684.512} C_VEL
LIN {X 0,Y 367.335,Z 478.624,A -85,B 0,C 180,E1 -12686.71,E2 -12686.71} C_VEL
LIN {X 0,Y 367.347,Z 479.785,A -85,B 0,C 180,E1 -12688.904,E2 -12688.904} C_VEL
LIN {X 0,Y 367.347,Z 479.782,A -85,B 0,C 180,E1 -12691.096,E2 -12691.096} C_VEL
LIN {X 0,Y 367.335,Z 478.612,A -85,B 0,C 180,E1 -12693.29,E2 -12693.29} C_VEL
LIN {X 0,Y 367.439,Z 476.297,A -85,B 0,C 180,E1 -12695.488,E2 -12695.488} C_VEL
LIN {X 0,Y 367.667,Z 472.785,A -85,B 0,C 180,E1 -12697.69,E2 -12697.69} C_VEL
LIN {X 0,Y 368.017,Z 467.987,A -85,B 0,C 180,E1 -12699.897,E2 -12699.897} C_VEL
LIN {X 0,Y 368.737,Z 461.774,A -85,B 0,C 180,E1 -12702.102,E2 -12702.102} C_VEL
LIN {X 0,Y 369.621,Z 453.969,A -85,B 0,C 180,E1 -12704.311,E2 -12704.311} C_VEL
LIN {X 0,Y 370.817,Z 445.669,A -85,B 0,C 180,E1 -12706.234,E2 -12706.234} C_VEL
LIN {X 0,Y 372.252,Z 435.666,A -85,B 0,C 180,E1 -12708.151,E2 -12708.151} C_VEL
LIN {X 0,Y 373.745,Z 425.434,A -85,B 0,C 180,E1 -12709.784,E2 -12709.784} C_VEL
LIN {X 0,Y 375.546,Z 413.24,A -85,B 0,C 180,E1 -12711.403,E2 -12711.403} C_VEL
LIN {X 0,Y 377.375,Z 399.658,A -85,B 0,C 180,E1 -12712.878,E2 -12712.878} C_VEL
LIN {X 0,Y 379.127,Z 386.038,A -85,B 0,C 180,E1 -12714.068,E2 -12714.068} C_VEL
LIN {X 0,Y 380.654,Z 371.923,A -85,B 0,C 180,E1 -12715.055,E2 -12715.055} C_VEL
LIN {X 0,Y 381.857,Z 358.055,A -85,B 0,C 180,E1 -12715.81,E2 -12715.81} C_VEL
LIN {X 0,Y 382.952,Z 342.47,A -85,B 0,C 180,E1 -12716.426,E2 -12716.426} C_VEL
LIN {X 0,Y 383.603,Z 327.145,A -85,B 0,C 180,E1 -12716.818,E2 -12716.818} C_VEL
LIN {X 0,Y 386.32,Z 212.136,A -85,B 0,C 180,E1 -12718.983,E2 -12718.983} C_VEL
LIN {X 0,Y 386.301,Z 207.072,A -85,B 0,C 180,E1 -12719.089,E2 -12719.089} C_VEL
LIN {X 0,Y 382.604,Z 188.322,A -85,B 0,C 180,E1 -12719.793,E2 -12719.793} C_VEL
LIN {X 0,Y 374.725,Z 170.855,A -85,B 0,C 180,E1 -12720.864,E2 -12720.864} C_VEL
LIN {X 0,Y 373.604,Z 168.188,A -85,B 0,C 180,E1 -12721.079,E2 -12721.079} C_VEL
LIN {X 0,Y 370.448,Z 155.774,A -85,B 0,C 180,E1 -12724.032,E2 -12724.032} C_VEL
LIN {X 0,Y 368.951,Z 150.243,A -85,B 0,C 180,E1 -12725.467,E2 -12725.467} C_VEL
LIN {X 0,Y 368.902,Z 150.143,A -85,B 0,C 180,E1 -12728.953,E2 -12728.953} C_VEL
LIN {X 0,Y 368.882,Z 150.159,A -85,B 0,C 180,E1 -12732.01,E2 -12732.01} C_VEL
LIN {X 0,Y 368.88,Z 150.15,A -85,B 0,C 180,E1 -12735.176,E2 -12735.176} C_VEL
LIN {X 0,Y 368.882,Z 150.142,A -85,B 0,C 180,E1 -12738.178,E2 -12738.178} C_VEL
LIN {X 0,Y 368.908,Z 150.145,A -85,B 0,C 180,E1 -12741.36,E2 -12741.36} C_VEL
LIN {X 0,Y 368.936,Z 150.127,A -85,B 0,C 180,E1 -12745.147,E2 -12745.147} C_VEL
LIN {X 0,Y 368.93,Z 150.133,A -85,B 0,C 180,E1 -12749.047,E2 -12749.047} C_VEL
LIN {X 0,Y 368.981,Z 150.149,A -85,B 0,C 180,E1 -12751.564,E2 -12751.564} C_VEL
LIN {X 0,Y 369.001,Z 150.132,A -85,B 0,C 180,E1 -12754.02,E2 -12754.02} C_VEL
LIN {X 0,Y 368.933,Z 150.147,A -85,B 0,C 180,E1 -12757.605,E2 -12757.605} C_VEL
LIN {X 0,Y 368.958,Z 150.151,A -85,B 0,C 180,E1 -12761.106,E2 -12761.106} C_VEL
LIN {X 0,Y 368.999,Z 150.13,A -85,B 0,C 180,E1 -12764.535,E2 -12764.535} C_VEL
LIN {X 0,Y 369.006,Z 150.143,A -85,B 0,C 180,E1 -12767.907,E2 -12767.907} C_VEL
LIN {X 0,Y 369.092,Z 150.122,A -85,B 0,C 180,E1 -12771.238,E2 -12771.238} C_VEL
LIN {X 0,Y 369.132,Z 150.123,A -85,B 0,C 180,E1 -12774.538,E2 -12774.538} C_VEL
LIN {X 0,Y 369.315,Z 150.096,A -85,B 0,C 180,E1 -12777.819,E2 -12777.819} C_VEL
LIN {X 0,Y 369.454,Z 150.087,A -85,B 0,C 180,E1 -12780,E2 -12780} C_VEL
LIN {X 0,Y 369.308,Z 150.089,A -85,B 0,C 180,E1 -12782.181,E2 -12782.181} C_VEL
LIN {X 0,Y 369.18,Z 150.118,A -85,B 0,C 180,E1 -12786.559,E2 -12786.559} C_VEL
LIN {X 0,Y 369.065,Z 150.127,A -85,B 0,C 180,E1 -12789.868,E2 -12789.868} C_VEL
LIN {X 0,Y 369.039,Z 150.128,A -85,B 0,C 180,E1 -12793.772,E2 -12793.772} C_VEL
LIN {X 0,Y 368.978,Z 150.15,A -85,B 0,C 180,E1 -12797.757,E2 -12797.757} C_VEL
LIN {X 0,Y 368.911,Z 150.148,A -85,B 0,C 180,E1 -12801.221,E2 -12801.221} C_VEL
LIN {X 0,Y 368.911,Z 150.15,A -85,B 0,C 180,E1 -12803.875,E2 -12803.875} C_VEL
LIN {X 0,Y 368.866,Z 150.16,A -85,B 0,C 180,E1 -12807.211,E2 -12807.211} C_VEL
LIN {X 0,Y 368.895,Z 150.142,A -85,B 0,C 180,E1 -12809.692,E2 -12809.692} C_VEL
LIN {X 0,Y 368.897,Z 150.114,A -85,B 0,C 180,E1 -12813.043,E2 -12813.043} C_VEL
LIN {X 0,Y 368.917,Z 150.157,A -85,B 0,C 180,E1 -12816.197,E2 -12816.197} C_VEL
LIN {X 0,Y 368.874,Z 150.132,A -85,B 0,C 180,E1 -12818.957,E2 -12818.957} C_VEL
LIN {X 0,Y 368.87,Z 150.146,A -85,B 0,C 180,E1 -12822.007,E2 -12822.007} C_VEL
LIN {X 0,Y 368.875,Z 150.145,A -85,B 0,C 180,E1 -12825.175,E2 -12825.175} C_VEL
LIN {X 0,Y 368.865,Z 150.163,A -85,B 0,C 180,E1 -12828.175,E2 -12828.175} C_VEL
LIN {X 0,Y 368.878,Z 150.155,A -85,B 0,C 180,E1 -12831.366,E2 -12831.366} C_VEL
LIN {X 0,Y 368.931,Z 150.158,A -85,B 0,C 180,E1 -12835.146,E2 -12835.146} C_VEL
LIN {X 0,Y 368.94,Z 150.269,A -85,B 0,C 180,E1 -12835.727,E2 -12835.727} C_VEL
LIN {X 0,Y 370.851,Z 157.527,A -85,B 0,C 180,E1 -12837.651,E2 -12837.651} C_VEL
LIN {X 0,Y 372.219,Z 162.717,A -85,B 0,C 180,E1 -12838.88,E2 -12838.88} C_VEL
LIN {X 0,Y 381.708,Z 183.262,A -85,B 0,C 180,E1 -12840.199,E2 -12840.199} C_VEL
LIN {X 0,Y 385.242,Z 192.144,A -85,B 0,C 180,E1 -12840.687,E2 -12840.687} C_VEL
LIN {X 0,Y 386.625,Z 199.551,A -85,B 0,C 180,E1 -12840.957,E2 -12840.957} C_VEL
LIN {X 0,Y 383.892,Z 313.263,A -85,B 0,C 180,E1 -12843.094,E2 -12843.094} C_VEL
LIN {X 0,Y 383.268,Z 332.481,A -85,B 0,C 180,E1 -12843.524,E2 -12843.524} C_VEL
LIN {X 0,Y 382.29,Z 347.954,A -85,B 0,C 180,E1 -12844.084,E2 -12844.084} C_VEL
LIN {X 0,Y 381.198,Z 362.561,A -85,B 0,C 180,E1 -12844.839,E2 -12844.839} C_VEL
LIN {X 0,Y 379.878,Z 375.49,A -85,B 0,C 180,E1 -12845.692,E2 -12845.692} C_VEL
LIN {X 0,Y 378.286,Z 388.438,A -85,B 0,C 180,E1 -12846.747,E2 -12846.747} C_VEL
LIN {X 0,Y 376.56,Z 401.674,A -85,B 0,C 180,E1 -12848.082,E2 -12848.082} C_VEL
LIN {X 0,Y 374.908,Z 413.505,A -85,B 0,C 180,E1 -12849.533,E2 -12849.533} C_VEL
